// 已中止 — 等待 Reset，支援 Resume
METHOD M_STATE_ABORTED
VAR_INPUT
END_VAR
IF NOT _bRetry THEN
	Busy 	:= FALSE;
	Aborted := TRUE;
	Error 	:= TRUE;
	Status 	:= strStatus;
	_AbortCompleted := FALSE;
	uiAbortingStep  := 0;
END_IF
// 等待上層 FB 設定 Reset
IF reset THEN
	_bRetry := TRUE;
	Busy 	:= FALSE;
	Aborted := FALSE;
	Error 	:= FALSE;
END_IF

IF NOT Execute THEN
	eState := STATE_RESETTING;
END_IF

IF Execute AND _bRetry AND NOT StorageRobot._DI1.Error AND NOT StorageRobot.Halt THEN
	status := '';
	uiExecutingStep := uiResumeStep;
	eState := STATE_EXECUTING;
END_IF
END_METHOD

// 中止 — 停止手臂/馬達/氣缸，保存 Resume 步驟
METHOD M_STATE_ABORTING
VAR_INPUT
END_VAR
CASE uiAbortingStep OF
0:
	// 保存 Resume
	IF uiResumeStep = 0 THEN
		uiResumeStep := uiExecutingStep;
	END_IF
	_Abort	:= FALSE;
	_bRetry := FALSE;

	// 清除 Timer
	TON_TimeOut.IN := FALSE;
	TON_ConveyorTimeOut.IN := FALSE;
	TON_RobotResetTimeOut.IN := FALSE;
	tonDelay_SameSizeGetBox.IN := FALSE;
	tonDelay_SameSizeDelayBox.IN := FALSE;
	uiSameGetBoxStep := 0;

	// 停止手臂 + 倉儲 + NG + PullOut
	//StorageRobot.M_ResetAllCommand();		續做盡量不要清除掉手臂的command 保持原狀，如要清除把Continue 拔掉即可。
	WareHouse.M_ResetFeedInBox();
	NGRegionMove.Execute := FALSE;
	PullOutRegionMove.Execute := FALSE;

	// Phase 2:清 local intent (A00 在 Busy 時 propagate FALSE,本 instance 收手不影響別人)
	bIntent_NeedBackward := FALSE;
	bIntent_HoldStill    := FALSE;

	uiAbortingStep := 100;

100:
	// 機構復位
	uiAbortingStep := 9999;
9999:
	_AbortCompleted := TRUE;
END_CASE

IF NOT Execute THEN
	estate := STATE_RESETTING;
ELSIF _AbortCompleted THEN
	eState := STATE_Aborted;
END_IF
END_METHOD

METHOD M_STATE_DONE
VAR_INPUT
END_VAR
Busy := FALSE;
Done := TRUE;

// 等待上層 FB 取消 Execute
IF NOT Execute THEN
	eState := STATE_RESETTING;
END_IF
END_METHOD

METHOD M_STATE_DORMANT
VAR_INPUT
END_VAR
Busy				:= FALSE;
Done				:= FALSE;
Aborted				:= FALSE;
Error				:= FALSE;
ErrorID				:= 0;
Status				:= '';
_ResetCompleted		:= FALSE;
_Error				:= FALSE;
_Executed			:= FALSE;
_Abort				:= FALSE;
uiExecutingStep		:= 0;
uiResettingStep		:= 0;
uiAbortingStep		:= 0;

_UniqueErrorCode	:= '';
_bRetry				:= FALSE;
uiResumeStep		:= 0;

bBoxA_Done			:= FALSE;
bBoxB_Done			:= FALSE;
bBoxReady			:= FALSE;
bDualGrip			:= FALSE;
bFirstClampIsA		:= TRUE;

TON_TimeOut.IN			:= FALSE;
TON_ConveyorTimeOut.IN	:= FALSE;
TON_RobotResetTimeOut.IN := FALSE;
TON_ArrivedDelay.IN		:= FALSE;
tonDelay_SameSizeGetBox.IN	:= FALSE;
tonDelay_SameSizeDelayBox.IN := FALSE;
uiSameGetBoxStep		:= 0;
tonErrorResetDelay.IN	:= FALSE;
bErrorBlinking			:= FALSE;

PullOutRegionMove.Execute := FALSE;
NGRegionMove.Execute      := FALSE;

// Phase 2:DORMANT 只清 local intent,不動 shared SameSizeCVRequest flag (本 FB 有兩個 instance,idle 不能 stomp 其他 instance 的 request)
bIntent_NeedBackward := FALSE;
bIntent_HoldStill    := FALSE;

_AbortCompleted		:= FALSE;

// 由上層 FB 設定 Execute := TRUE 觸發
IF Execute AND NOT Stop THEN
	// 啟動前檢查
	IF NOT bBoxA_Enable AND NOT bBoxB_Enable THEN
		strStatus := 'No box enabled';
		_UniqueErrorCode := 'E_NO_BOX';
		_Abort := TRUE;
		RETURN;
	END_IF

	// 判斷爪模式
	bDualGrip := bBoxA_Enable AND bBoxB_Enable;
	IF bBoxA_Enable THEN
		bFirstClampIsA := TRUE;
	ELSIF bBoxB_Enable THEN
		bFirstClampIsA := FALSE;
	END_IF

	eState := STATE_EXECUTING;
END_IF
END_METHOD

METHOD M_STATE_ERROR
VAR_INPUT
END_VAR
Busy := FALSE;
Error := TRUE;
Status := strStatus;

// Reset 上升緣 → 1 秒閃爍 (對齊 FB_ShippingRobotTransfer)
trigErrorReset(CLK := Reset);
IF trigErrorReset.Q THEN
	bErrorBlinking := TRUE;
END_IF
tonErrorResetDelay(IN := bErrorBlinking, PT := T#1S);
IF tonErrorResetDelay.Q THEN
	bErrorBlinking := FALSE;
END_IF
IF bErrorBlinking THEN
	Error := FALSE;
END_IF

IF NOT Execute THEN
	Error := FALSE;
	bErrorBlinking := FALSE;
	tonErrorResetDelay.IN := FALSE;
	eState := STATE_RESETTING;
ELSIF trigErrorReset.Q AND Execute AND NOT StorageRobot._DI1.Error THEN
	// Retry 對稱:Reset 上升緣 (edge) 才觸發,從 uiResumeStep 續做
	uiExecutingStep := uiResumeStep;
	Status := '';
	Error := FALSE;
	bErrorBlinking := FALSE;
	tonErrorResetDelay.IN := FALSE;
	eState := STATE_EXECUTING;
END_IF
END_METHOD

// 執行主狀態 — 軌道送盒 + 大手臂取盒 + 入倉/NG
// ═══════════════════════════════════════════════════
// Phase 1 (1000-1500): 第一盒送到 NearStorage
// Phase 2 (2000-2100): 大手臂取第一盒
// Phase 3 (3000-3400): 第二盒送到 NearStorage (雙爪)
// Phase 4 (4000-4100): 大手臂取第二盒
// Phase 5 (5000-5600): 放 ClampA (入倉 or NG)
// Phase 6 (6000-6500): 放 ClampB (入倉 or NG)
// Phase 9 (9000-9100): 復位機構
// ═══════════════════════════════════════════════════
METHOD M_STATE_EXECUTING
VAR_INPUT
END_VAR
Busy := TRUE;

// Stop 時暫停 Timeout
IF Stop THEN
	TON_TimeOut.IN := FALSE;
	TON_ConveyorTimeOut.IN := FALSE;
END_IF

CASE uiExecutingStep OF

0:	// 初始化
	bBoxReady := FALSE;
	bBoxA_Done := FALSE;
	bBoxB_Done := FALSE;
	uiExecutingStep := 1000;

{region '=== Phase 1: 第一盒送到 NearStorage ==='}
// 流程: 馬達 backward + 擋盒 state machine (Press3 後壓 + Press4 擋第二盒) → 送到 NearStorage → motor 停
// 擋盒邏輯 ref FB_RobotRegionMove_AllocatedConveyor uiSameGetBoxStep 0/100/200/300/400 (省略 325/350/375 卡盒重推,Reverse 流程 motor 不能 forward)

1000:	// 請求軌道 backward + 初始化擋盒 state machine
	bIntent_NeedBackward := TRUE;
	bIntent_HoldStill    := FALSE;
	Cylinder.List.fbSameSizeCV_Press3.M_Retract();
	Cylinder.List.fbSameSizeCV_Press4.M_Retract();
	uiSameGetBoxStep := 0;
	TON_ConveyorTimeOut.IN := TRUE;
	uiExecutingStep := 1100;

1100:	// 擋盒 state machine
	CASE uiSameGetBoxStep OF
		0:	// 初始位置:兩支 retract
			Cylinder.List.fbSameSizeCV_Press3.M_Retract();
			Cylinder.List.fbSameSizeCV_Press4.M_Retract();
			uiSameGetBoxStep := 100;

		100:	// 等盒到 Detect6 (50ms debounce) → Press3 extend 後壓
			tonDelay_SameSizeGetBox.IN := Input.bSameSizeCV_BoxDetect6_Sensor;
			IF tonDelay_SameSizeGetBox.Q THEN
				Cylinder.List.fbSameSizeCV_Press3.M_Extend();
				uiSameGetBoxStep := 200;
			END_IF

		200:	// 等 NearStorageSensor 穩定 1.5s 確認盒到位
			tonDelay_SameSizeGetBox.IN := FALSE;
			tonDelay_SameSizeDelayBox.IN := Input.bSameSizeCV_BoxNearStorageSensor;
			IF tonDelay_SameSizeDelayBox.Q THEN
				uiSameGetBoxStep := 300;
			END_IF

		300:	// Press4 extend 擋第二盒避免擠進來
			Cylinder.List.fbSameSizeCV_Press4.M_Extend();
			IF Cylinder.List.fbSameSizeCV_Press4.InFrontPosition THEN
				uiSameGetBoxStep := 400;
			END_IF

		400:	// state machine 完成 → 進 1500 motor 停 + final settle
			tonDelay_SameSizeDelayBox.IN := FALSE;
			uiSameGetBoxStep := 0;
			TON_ConveyorTimeOut.IN := FALSE;
			uiExecutingStep := 1500;
	END_CASE
	// state machine 整段 60s timeout 保護
	IF TON_ConveyorTimeOut.Q THEN
		TON_ConveyorTimeOut.IN := FALSE;
		uiResumeStep := 1000;
		strStatus := 'Phase 1 擋盒 state machine timeout';
		_UniqueErrorCode := 'E_BLOCK_TIMEOUT';
		_Abort := TRUE;
	END_IF

1500:	// 軌道 backward 推到 NearStorage final settle (Press3 後壓中, Press4 擋第二盒中)
	TON_ConveyorTimeOut.IN := TRUE;
	TON_ArrivedDelay.IN := Input.bSameSizeCV_BoxNearStorageSensor;
	IF TON_ArrivedDelay.Q THEN
		TON_ConveyorTimeOut.IN := FALSE;
		bIntent_NeedBackward := FALSE;
		bIntent_HoldStill    := TRUE;	// 大手臂取盒前要靜止
		uiExecutingStep := 1600;
	END_IF
	IF TON_ConveyorTimeOut.Q THEN
		bIntent_NeedBackward := FALSE;
		uiResumeStep := 1000;	// retry 從馬達啟動重來
		strStatus := 'Box cross conveyor timeout';
		_UniqueErrorCode := 'E_BOX_CROSS_TIMEOUT';
		_Abort := TRUE;
	END_IF

1600:	// 等待馬達停止
	 TON_ArrivedDelay.IN := FALSE;
	IF Motor.List.TransmitSameSideCV.InStopped THEN
		//uiExecutingStep := 1650;
		uiExecutingStep := 2000;
	END_IF
1650:	// dead code (1600 直接跳 2000),保留以維持原邏輯 — Destination=WareHouse 視同舊 IsOK=TRUE
	 IF eBoxA_Destination = E_ReverseBoxDestination.WareHouse THEN
	  	uiExecutingStep := 2000;
	 ELSE
		uiExecutingStep := 1700;
  	 END_IF
	 
1700:
	TON_TimeOut.IN := TRUE;
	Cylinder.List.fbSameSizeCV_Press4.M_Extend();
	IF Cylinder.List.fbSameSizeCV_Press4.InFrontPosition THEN
		TON_TimeOut.IN := FALSE;
		uiExecutingStep := 1800;
	END_IF
	IF TON_TimeOut.Q THEN
		uiResumeStep := uiExecutingStep;
		strStatus := 'Press4 Extend timeout';
		_UniqueErrorCode := 'E_CYL_TIMEOUT';
		_Abort := TRUE;
	END_IF
1800:
	Cylinder.List.fbSameSizeCV_Press4.M_Retract();
	IF Cylinder.List.fbSameSizeCV_Press4.InRearPosition THEN				
		uiExecutingStep := 2000;
	END_IF
		 
{endregion}

{region '=== Phase 2: 大手臂取第一盒 ==='}

2000:	// Robot AbsMove 取盒
	TON_TimeOut.IN := TRUE;
	IF NOT StorageRobot._DI1.Done THEN
		StorageRobot.M_StartRobotAbsMove(
			GetBox			:= TRUE,
			UseClampA		:= bFirstClampIsA,
			UseClampB		:= FALSE,
			Area			:= E_RobotArea.TransmitCV,
			ClampA_Address	:= PickupPosition,
			ClampB_Address	:= 99,
			BoxReady_1		:= bFirstClampIsA,
			BoxReady_2		:= FALSE);
	ELSE
		TON_TimeOut.IN := FALSE;
		uiExecutingStep := 2100;
	END_IF
	IF TON_TimeOut.Q OR StorageRobot.Error THEN
		uiResumeStep := uiExecutingStep;
		strStatus := 'Robot pick first box timeout';
		_UniqueErrorCode := 'E_BIGARM_TIMEOUT';
		_Abort := TRUE;
	END_IF

2100:	// Reset Robot
	StorageRobot.M_ResetAllCommand();
	IF NOT StorageRobot._DI1.Done THEN
		IF bDualGrip THEN
			uiExecutingStep := 3000;
		ELSE
			uiExecutingStep := 5000;
		END_IF
	END_IF

{endregion}

{region '=== Phase 3: 第二盒送到 NearStorage (雙爪) ==='}
// 流程同 Phase 1:馬達 backward + 擋盒 state machine → 送到 NearStorage → motor 停

3000:	// 請求軌道 backward + 初始化擋盒 state machine (第二盒)
	bIntent_NeedBackward := TRUE;
	bIntent_HoldStill    := FALSE;
	Cylinder.List.fbSameSizeCV_Press3.M_Retract();
	Cylinder.List.fbSameSizeCV_Press4.M_Retract();
	uiSameGetBoxStep := 0;
	TON_ConveyorTimeOut.IN := TRUE;
	uiExecutingStep := 3100;

3100:	// 擋盒 state machine (第二盒) — ref AllocatedConveyor (與 Phase 1 step 1100 對稱)
	CASE uiSameGetBoxStep OF
		0:
			Cylinder.List.fbSameSizeCV_Press3.M_Retract();
			Cylinder.List.fbSameSizeCV_Press4.M_Retract();
			uiSameGetBoxStep := 100;

		100:	// 等盒到 Detect6 (50ms debounce) → Press3 extend
			tonDelay_SameSizeGetBox.IN := Input.bSameSizeCV_BoxDetect6_Sensor;
			IF tonDelay_SameSizeGetBox.Q THEN
				Cylinder.List.fbSameSizeCV_Press3.M_Extend();
				uiSameGetBoxStep := 200;
			END_IF

		200:	// 等 NearStorageSensor 穩定 1.5s
			tonDelay_SameSizeGetBox.IN := FALSE;
			tonDelay_SameSizeDelayBox.IN := Input.bSameSizeCV_BoxNearStorageSensor;
			IF tonDelay_SameSizeDelayBox.Q THEN
				uiSameGetBoxStep := 300;
			END_IF

		300:	// Press4 extend
			Cylinder.List.fbSameSizeCV_Press4.M_Extend();
			IF Cylinder.List.fbSameSizeCV_Press4.InFrontPosition THEN
				uiSameGetBoxStep := 400;
			END_IF

		400:	// 完成 → 進 3500
			tonDelay_SameSizeDelayBox.IN := FALSE;
			uiSameGetBoxStep := 0;
			TON_ConveyorTimeOut.IN := FALSE;
			uiExecutingStep := 3500;
	END_CASE
	IF TON_ConveyorTimeOut.Q THEN
		TON_ConveyorTimeOut.IN := FALSE;
		uiResumeStep := 3000;
		strStatus := 'Phase 3 擋盒 state machine timeout';
		_UniqueErrorCode := 'E_BLOCK_TIMEOUT';
		_Abort := TRUE;
	END_IF

3500:	// 軌道 backward 推到 NearStorage final settle (第二盒)
	TON_ConveyorTimeOut.IN := TRUE;
	TON_ArrivedDelay.IN := Input.bSameSizeCV_BoxNearStorageSensor;
	IF TON_ArrivedDelay.Q THEN
		TON_ConveyorTimeOut.IN := FALSE;
		bIntent_NeedBackward := FALSE;
		bIntent_HoldStill    := TRUE;	// 大手臂取盒前要靜止
		uiExecutingStep := 3600;
	END_IF
	IF TON_ConveyorTimeOut.Q THEN
		bIntent_NeedBackward := FALSE;
		uiResumeStep := 3000;	// retry 從馬達啟動重來
		strStatus := 'Box 2 cross conveyor timeout';
		_UniqueErrorCode := 'E_BOX_CROSS_TIMEOUT';
		_Abort := TRUE;
	END_IF

3600:	// 等待馬達停止
	 TON_ArrivedDelay.IN := FALSE;
	IF Motor.List.TransmitSameSideCV.InStopped THEN
		//uiExecutingStep := 3650;
		uiExecutingStep := 4000;
	END_IF
3650:	// dead code,保留 — Destination=WareHouse 視同舊 IsOK=TRUE
	 IF eBoxB_Destination = E_ReverseBoxDestination.WareHouse THEN
	  	uiExecutingStep := 4000;
	 ELSE
		uiExecutingStep := 3700;
  	 END_IF
	 
3700:
	TON_TimeOut.IN := TRUE;
	Cylinder.List.fbSameSizeCV_Press4.M_Extend();
	IF Cylinder.List.fbSameSizeCV_Press4.InFrontPosition THEN
		TON_TimeOut.IN := FALSE;
		uiExecutingStep := 3800;
	END_IF
	IF TON_TimeOut.Q THEN
		uiResumeStep := uiExecutingStep;
		strStatus := 'Press4 Extend timeout';
		_UniqueErrorCode := 'E_CYL_TIMEOUT';
		_Abort := TRUE;
	END_IF
3800:
	Cylinder.List.fbSameSizeCV_Press4.M_Retract();
	IF Cylinder.List.fbSameSizeCV_Press4.InRearPosition THEN				
		uiExecutingStep := 4000;
	END_IF

{endregion}

{region '=== Phase 4: 大手臂取第二盒 ==='}

4000:	// Robot AbsMove 第二爪
	TON_TimeOut.IN := TRUE;
	IF NOT StorageRobot._DI1.Done THEN
		StorageRobot.M_StartRobotAbsMove(
			GetBox			:= TRUE,
			UseClampA		:= FALSE,
			UseClampB		:= bFirstClampIsA,
			Area			:= E_RobotArea.TransmitCV,
			ClampA_Address	:= 99,
			ClampB_Address	:= PickupPosition,
			BoxReady_1		:= FALSE,
			BoxReady_2		:= bFirstClampIsA);
	ELSE
		TON_TimeOut.IN := FALSE;
		uiExecutingStep := 4100;
	END_IF
	IF TON_TimeOut.Q OR StorageRobot.Error THEN
		uiResumeStep := uiExecutingStep;
		strStatus := 'Robot pick second box timeout';
		_UniqueErrorCode := 'E_BIGARM_TIMEOUT';
		_Abort := TRUE;
	END_IF

4100:	// Reset Robot
	StorageRobot.M_ResetAllCommand();
	IF NOT StorageRobot._DI1.Done THEN
		uiExecutingStep := 5000;
	END_IF

{endregion}

{region '=== Phase 5: 放 ClampA ==='}

5000:	// 清除 Robot 命令
	TON_RobotResetTimeOut.IN := TRUE;
	StorageRobot.M_ResetAllCommand();
	IF NOT StorageRobot._DI1.Done AND
		NOT (StorageRobot._DI1.AbsMoveA OR StorageRobot._DI1.AbsMoveB OR
			 StorageRobot._DI1.WarehouseA OR StorageRobot._DI1.WarehouseB) THEN
		TON_RobotResetTimeOut.IN := FALSE;
		bBoxReady := FALSE;
		IF bBoxA_Enable THEN
			uiExecutingStep := 5100;
		ELSE
			uiExecutingStep := 6000;
		END_IF
	END_IF
	IF TON_RobotResetTimeOut.Q THEN
		uiResumeStep := 5000;
		strStatus := 'Robot reset timeout (phase 5)';
		_UniqueErrorCode := 'E_BIGARM_TIMEOUT';
		_Abort := TRUE;
	END_IF

5100:	// ClampA Destination 三選一
	CASE eBoxA_Destination OF
		E_ReverseBoxDestination.WareHouse:
			uiExecutingStep := 5200;
		E_ReverseBoxDestination.PullOut:
			uiExecutingStep := 5400;
		E_ReverseBoxDestination.NGConveyor:
			uiExecutingStep := 5300;
	ELSE
		uiResumeStep := 5100;
		strStatus := 'Invalid BoxA destination enum';
		_UniqueErrorCode := 'E_INVALID_DEST';
		_Abort := TRUE;
	END_CASE

5200:	// ClampA OK → 入倉
	TON_TimeOut.IN := TRUE;
	stWareHouseCoord.Layer := iBoxA_Level;
	stWareHouseCoord.Slide := iBoxA_Track;
	IF iBoxA_Warehouse = 1 THEN
		WareHouse.M_StartFeedInBox(WareHouseSelect := E_WareHouse.WareHouseA, WarehouseCoordinates := stWareHouseCoord);
		IF WareHouse.bFeedInBox_Completed THEN
			bBoxReady := TRUE;
		END_IF
		StorageRobot.M_StartWareHousePlaceBox_ClampA(
			WareHouseSelect := E_WareHouse.WareHouseA,
			Info := stWareHouseCoord,
			BoxReady_1st := bBoxReady);
	ELSIF iBoxA_Warehouse = 2 THEN
		WareHouse.M_StartFeedInBox(WareHouseSelect := E_WareHouse.WareHouseB, WarehouseCoordinates := stWareHouseCoord);
		IF WareHouse.bFeedInBox_Completed THEN
			bBoxReady := TRUE;
		END_IF
		StorageRobot.M_StartWareHousePlaceBox_ClampA(
			WareHouseSelect := E_WareHouse.WareHouseB,
			Info := stWareHouseCoord,
			BoxReady_1st := bBoxReady);
	ELSE
		uiResumeStep := 5200;
		strStatus := 'Invalid BoxA warehouse value';
		_UniqueErrorCode := 'E_INVALID_WAREHOUSE';
		_Abort := TRUE;
		RETURN;
	END_IF
	IF StorageRobot._DI1.Done THEN
		TON_TimeOut.IN := FALSE;
		bBoxA_Done := TRUE;
		uiExecutingStep := 5500;
	END_IF
	IF TON_TimeOut.Q OR StorageRobot.Error THEN
		uiResumeStep := 5200;
		strStatus := 'ClampA place to warehouse timeout';
		_UniqueErrorCode := 'E_BIGARM_TIMEOUT';
		_Abort := TRUE;
	END_IF

5300:	// ClampA NG → NG區
	NGRegionMove.Info.Get := FALSE;
	NGRegionMove.Info.UseA := TRUE;
	NGRegionMove.Info.UseB := FALSE;
	NGRegionMove.Info.A_Position := NGAreaPosition;
	NGRegionMove.Info.B_Position := 0;
	NGRegionMove.Execute := TRUE;
	uiExecutingStep := 5310;

5310:	// 等待 NG RegionMove 完成
	IF NGRegionMove.Done THEN
		NGRegionMove.Execute := FALSE;
		bBoxA_Done := TRUE;
		uiExecutingStep := 5320;
	END_IF
	IF NGRegionMove.Error OR NGRegionMove.Aborted THEN
		NGRegionMove.Execute := FALSE;
		uiResumeStep := 5300;
		strStatus := 'ClampA NG region move failed';
		_UniqueErrorCode := 'E_BIGARM_TIMEOUT';
		_Abort := TRUE;
	END_IF

5320:	// 等待 DORMANT
	IF NOT NGRegionMove.Busy AND NOT NGRegionMove.Done THEN
		uiExecutingStep := 5600;
	END_IF

5400:	// ClampA PullOut → PullOutConveyor 區 (Side 1=I3_Slide 左, 2=I4_Slide 右)
	IF iBoxA_PullOutSide < 1 OR iBoxA_PullOutSide > 2 THEN
		uiResumeStep := 5400;
		strStatus := 'Invalid BoxA PullOut side (must be 1 or 2)';
		_UniqueErrorCode := 'E_INVALID_PULLOUT_SIDE';
		_Abort := TRUE;
	ELSE
		PullOutRegionMove.Info.Get := FALSE;
		PullOutRegionMove.Info.UseA := TRUE;
		PullOutRegionMove.Info.UseB := FALSE;
		PullOutRegionMove.Info.A_Position := iBoxA_PullOutSide;
		PullOutRegionMove.Info.B_Position := 0;
		PullOutRegionMove.Execute := TRUE;
		uiExecutingStep := 5410;
	END_IF

5410:	// 等待 PullOut RegionMove 完成
	IF PullOutRegionMove.Done THEN
		PullOutRegionMove.Execute := FALSE;
		bBoxA_Done := TRUE;
		uiExecutingStep := 5420;
	END_IF
	IF PullOutRegionMove.Error OR PullOutRegionMove.Aborted THEN
		PullOutRegionMove.Execute := FALSE;
		uiResumeStep := 5400;
		strStatus := 'ClampA PullOut region move failed';
		_UniqueErrorCode := 'E_BIGARM_TIMEOUT';
		_Abort := TRUE;
	END_IF

5420:	// 等待 DORMANT
	IF NOT PullOutRegionMove.Busy AND NOT PullOutRegionMove.Done THEN
		uiExecutingStep := 5600;
	END_IF

5500:	// ClampA OK 完成 → Reset
	StorageRobot.M_ResetAllCommand();
	WareHouse.M_ResetFeedInBox();
	IF NOT StorageRobot._DI1.Done THEN
		uiExecutingStep := 5600;
	END_IF

5600:	// 繼續 ClampB?
	IF bDualGrip THEN
		bBoxReady := FALSE;
		uiExecutingStep := 6000;
	ELSE
		uiExecutingStep := 9000;
	END_IF

{endregion}

{region '=== Phase 6: 放 ClampB ==='}

6000:	// 準備放 ClampB
	TON_RobotResetTimeOut.IN := TRUE;
	StorageRobot.M_ResetAllCommand();
	IF NOT StorageRobot._DI1.Done AND
		NOT (StorageRobot._DI1.AbsMoveA OR StorageRobot._DI1.AbsMoveB OR
			 StorageRobot._DI1.WarehouseA OR StorageRobot._DI1.WarehouseB) THEN
		TON_RobotResetTimeOut.IN := FALSE;
		uiExecutingStep := 6100;
	END_IF
	IF TON_RobotResetTimeOut.Q THEN
		uiResumeStep := 6000;
		strStatus := 'Robot reset timeout (phase 6)';
		_UniqueErrorCode := 'E_BIGARM_TIMEOUT';
		_Abort := TRUE;
	END_IF

6100:	// ClampB Destination 三選一
	CASE eBoxB_Destination OF
		E_ReverseBoxDestination.WareHouse:
			uiExecutingStep := 6200;
		E_ReverseBoxDestination.PullOut:
			uiExecutingStep := 6400;
		E_ReverseBoxDestination.NGConveyor:
			uiExecutingStep := 6300;
	ELSE
		uiResumeStep := 6100;
		strStatus := 'Invalid BoxB destination enum';
		_UniqueErrorCode := 'E_INVALID_DEST';
		_Abort := TRUE;
	END_CASE

6200:	// ClampB OK → 入倉
	TON_TimeOut.IN := TRUE;
	stWareHouseCoord.Layer := iBoxB_Level;
	stWareHouseCoord.Slide := iBoxB_Track;
	IF iBoxB_Warehouse = 1 THEN
		WareHouse.M_StartFeedInBox(WareHouseSelect := E_WareHouse.WareHouseA, WarehouseCoordinates := stWareHouseCoord);
		IF WareHouse.bFeedInBox_Completed THEN
			bBoxReady := TRUE;
		END_IF
		StorageRobot.M_StartWareHousePlaceBox_ClampB(
			WareHouseSelect := E_WareHouse.WareHouseA,
			Info := stWareHouseCoord,
			BoxReady_2nd := bBoxReady);
	ELSIF iBoxB_Warehouse = 2 THEN
		WareHouse.M_StartFeedInBox(WareHouseSelect := E_WareHouse.WareHouseB, WarehouseCoordinates := stWareHouseCoord);
		IF WareHouse.bFeedInBox_Completed THEN
			bBoxReady := TRUE;
		END_IF
		StorageRobot.M_StartWareHousePlaceBox_ClampB(
			WareHouseSelect := E_WareHouse.WareHouseB,
			Info := stWareHouseCoord,
			BoxReady_2nd := bBoxReady);
	ELSE
		uiResumeStep := 6200;
		strStatus := 'Invalid BoxB warehouse value';
		_UniqueErrorCode := 'E_INVALID_WAREHOUSE';
		_Abort := TRUE;
		RETURN;
	END_IF
	IF StorageRobot._DI1.Done THEN
		TON_TimeOut.IN := FALSE;
		bBoxB_Done := TRUE;
		uiExecutingStep := 6500;
	END_IF
	IF TON_TimeOut.Q OR StorageRobot.Error THEN
		uiResumeStep := 6200;
		strStatus := 'ClampB place to warehouse timeout';
		_UniqueErrorCode := 'E_BIGARM_TIMEOUT';
		_Abort := TRUE;
	END_IF

6300:	// ClampB NG → NG區
	NGRegionMove.Info.Get := FALSE;
	NGRegionMove.Info.UseA := FALSE;
	NGRegionMove.Info.UseB := TRUE;
	NGRegionMove.Info.A_Position := 0;
	NGRegionMove.Info.B_Position := NGAreaPosition;
	NGRegionMove.Execute := TRUE;
	uiExecutingStep := 6310;

6310:	// 等待 NG 完成
	IF NGRegionMove.Done THEN
		NGRegionMove.Execute := FALSE;
		bBoxB_Done := TRUE;
		uiExecutingStep := 6320;
	END_IF
	IF NGRegionMove.Error OR NGRegionMove.Aborted THEN
		NGRegionMove.Execute := FALSE;
		uiResumeStep := 6300;
		strStatus := 'ClampB NG region move failed';
		_UniqueErrorCode := 'E_BIGARM_TIMEOUT';
		_Abort := TRUE;
	END_IF

6320:	// 等待 DORMANT
	IF NOT NGRegionMove.Busy AND NOT NGRegionMove.Done THEN
		uiExecutingStep := 9000;
	END_IF

6400:	// ClampB PullOut → PullOutConveyor 區 (Side 1=I3_Slide 左, 2=I4_Slide 右)
	IF iBoxB_PullOutSide < 1 OR iBoxB_PullOutSide > 2 THEN
		uiResumeStep := 6400;
		strStatus := 'Invalid BoxB PullOut side (must be 1 or 2)';
		_UniqueErrorCode := 'E_INVALID_PULLOUT_SIDE';
		_Abort := TRUE;
	ELSE
		PullOutRegionMove.Info.Get := FALSE;
		PullOutRegionMove.Info.UseA := FALSE;
		PullOutRegionMove.Info.UseB := TRUE;
		PullOutRegionMove.Info.A_Position := 0;
		PullOutRegionMove.Info.B_Position := iBoxB_PullOutSide;
		PullOutRegionMove.Execute := TRUE;
		uiExecutingStep := 6410;
	END_IF

6410:	// 等待 PullOut 完成
	IF PullOutRegionMove.Done THEN
		PullOutRegionMove.Execute := FALSE;
		bBoxB_Done := TRUE;
		uiExecutingStep := 6420;
	END_IF
	IF PullOutRegionMove.Error OR PullOutRegionMove.Aborted THEN
		PullOutRegionMove.Execute := FALSE;
		uiResumeStep := 6400;
		strStatus := 'ClampB PullOut region move failed';
		_UniqueErrorCode := 'E_BIGARM_TIMEOUT';
		_Abort := TRUE;
	END_IF

6420:	// 等待 DORMANT
	IF NOT PullOutRegionMove.Busy AND NOT PullOutRegionMove.Done THEN
		uiExecutingStep := 9000;
	END_IF

6500:	// ClampB OK 完成 → Reset
	StorageRobot.M_ResetAllCommand();
	WareHouse.M_ResetFeedInBox();
	IF NOT StorageRobot._DI1.Done THEN
		uiExecutingStep := 9000;
	END_IF

{endregion}

{region '=== Phase 9: 復位 ==='}

9000:	// 復位機構 (Phase 2:清 local intent,Busy 仍 TRUE 時 A00 會 propagate FALSE)
	bIntent_NeedBackward := FALSE;
	bIntent_HoldStill    := FALSE;
	Cylinder.List.fbSameSizeCV_Press3.M_Retract();
	Cylinder.List.fbSameSizeCV_Press4.M_Retract();
	uiExecutingStep := 9100;

9100:	// 等待復位完成 (Press3 + Press4 縮回 + 馬達停)
	TON_TimeOut.IN := TRUE;
	IF Cylinder.List.fbSameSizeCV_Press3.InRearPosition AND
	   Cylinder.List.fbSameSizeCV_Press4.InRearPosition AND
	   Motor.List.TransmitSameSideCV.InStopped THEN
		TON_TimeOut.IN := FALSE;
		_Executed := TRUE;
	END_IF
	IF TON_TimeOut.Q THEN
		uiResumeStep := uiExecutingStep;
		strStatus := 'Mechanism reset timeout';
		_UniqueErrorCode := 'E_CYL_TIMEOUT';
		_Abort := TRUE;
	END_IF

{endregion}

END_CASE

// 狀態切換
IF _Error THEN
	eState := STATE_ERROR;
ELSIF _Abort THEN
	eState := STATE_ABORTING;
ELSIF _Executed THEN
	eState := STATE_DONE;
ELSIF NOT Execute THEN
	eState := STATE_RESETTING; 
END_IF
END_METHOD

METHOD M_STATE_RESETTING
VAR_INPUT
END_VAR
Busy := TRUE;
Error := FALSE;
Aborted := FALSE;

CASE uiResettingStep OF
0:
	TON_TimeOut.IN := FALSE;
	TON_ConveyorTimeOut.IN := FALSE;
	TON_RobotResetTimeOut.IN := FALSE;
	tonDelay_SameSizeGetBox.IN := FALSE;
	tonDelay_SameSizeDelayBox.IN := FALSE;
	uiSameGetBoxStep := 0;

	StorageRobot.M_ResetAllCommand();
	WareHouse.M_ResetFeedInBox();
	NGRegionMove.Execute := FALSE;
	PullOutRegionMove.Execute := FALSE;
	// Phase 2:清 local intent (Busy=FALSE A00 不會寫,不影響別 instance shared flag)
	bIntent_NeedBackward := FALSE;
	bIntent_HoldStill    := FALSE;

	uiResettingStep := 100;

100:
	Done := FALSE;
	Busy := FALSE;
	_ResetCompleted := TRUE;
END_CASE

IF _ResetCompleted THEN
	eState := STATE_DORMANT;
END_IF
END_METHOD

END_FUNCTION_BLOCK

// ---- Library/20_MachineUnits/22_AllocateArea/Service/FB_PullOutConveyorAction.TcPOU
FUNCTION_BLOCK FB_PullOutConveyorAction EXTENDS FB_ObjectBase_V2 IMPLEMENTS IBasicElement
VAR_INPUT
    FixCylinderA1    : REFERENCE TO FB_Cylinder; // Conveyor A-side 1st cylinder
    FixCylinderA2    : REFERENCE TO FB_Cylinder; // Conveyor A-side 2nd cylinder
    FixCylinderB1    : REFERENCE TO FB_Cylinder; // Conveyor B-side 1st cylinder
    FixCylinderB2    : REFERENCE TO FB_Cylinder; // Conveyor B-side 2nd cylinder
    BarrierCylinderA : REFERENCE TO FB_Cylinder; // Conveyor A-side Barrier cylinder
    BarrierCylinderB : REFERENCE TO FB_Cylinder; // Conveyor B-side Barrier cylinder
    ConveyorMotorA    : REFERENCE TO FB_Motor; // PullOut Conveyor Motor 
	ConveyorMotorB	 : REFERENCE TO FB_Motor; //  Add New Motor Iomapping  edit Min 20250408
	INPUT            : REFERENCE TO ST_InputTable;	
    PullOutInfo      : ST_PullOutConveyorInfo;
END_VAR
VAR_OUTPUT
END_VAR
VAR
	FeedInSensor_A   : BOOL; // PullOut Conveyor A-side FeedIn Sensor
    FeedOutSensor_A  : BOOL; // PullOut Conveyor A-side FeedOut sensor
    DetactSensor_A   : BOOL; // PullOut Conveyor A-side detact sensor
    FeedInSensor_B   : BOOL; // PullOut Conveyor B-side FeedIn Sensor
    FeedOutSensor_B  : BOOL; // PullOut Conveyor B-side FeedOut sensor
    DetactSensor_B   : BOOL; // PullOut Conveyor B-side detact sensor
    TON_MotorRun     : TON; // Pull out conveyor motor running timer.
	TON_MotorReverse : TON; // Pull out conveyor motor reverse timer.
    TON_ForceForward : TON; // When auto process on, the time of force running in command direction.
	TON_MotorStopDelay : TON; // When Conveyor motor stop, the motor will be stopped later, so we need to give a time delay. 
    TON_BoxArrivedDelay: TON; // Check Box arrived(BoxA and BoxB) and delay.
	TON_BarryDelay : TON;
	tonFeedOutTimeOut :TON;
	tonMotorBReverse :TON;
	tonSensorDetectDelay : TON;
	TON_FeedInsensorADelay	:TON;
	TON_betweenboxReverse 	:TON;
	TON_PullOutTimeOut		:TON;
//	_Abort           : BOOL;
	bError			 : BOOL;
	strStatus	     : STRING;
	_UniqueErrorCode : STRING;
	PreviousStrStatus : STRING;
	PreviousErrorCode : STRING;
	
	uiResumeStep	: UINT;
	_bRetry	: BOOL;
END_VAR

A00_BasicUnits();
A10_StateControl();

ACTION A00_BasicUnits:
TON_MotorRun		(PT	:= PullOutInfo.ConveyorRunningTime);
TON_MotorReverse	(PT	:= PullOutInfo.ConveyorReverseTime);
TON_ForceForward	(PT	:= T#0.5S);
TON_MotorStopDelay	(PT := PullOutInfo.ConveyorReverseTime);
TON_BoxArrivedDelay	(PT := T#800MS);
TON_BarryDelay		(PT	:= T#0.1S);
tonFeedOutTimeOut	(PT := PullOutInfo.ConveyorReverseTime*3 );		//notthing use
tonMotorBReverse	(PT := T#1.5S);


tonSensorDetectDelay(PT	:= T#100MS);
TON_FeedInsensorADelay(PT :=T#700MS);
TON_betweenboxReverse(PT :=T#700MS);
TON_PullOutTimeOut (PT :=T#20.0S);



ErrorID := GVL_ErrorCode.GC_SVCID_ALC_PULLOUT_CV;
END_ACTION

ACTION A01_clcExecuting:
FeedInSensor_A  :=INPUT.bPullOutCV_AsideEntry_Sensor;
FeedOutSensor_A  :=INPUT.bPullOutCV_AsideExit_Sensor;
DetactSensor_A   :=input.bPullOutCV_Aside2ndBoxGap_Sensor;
FeedInSensor_B   :=INPUT.bPullOutCV_BsideEntry_Sensor;
FeedOutSensor_B  := INPUT.bPullOutCV_BsideExit_Sensor;
DetactSensor_B   := INPUT.bPullOutCV_Bside2ndBoxGap_Sensor;
END_ACTION

METHOD M_CheckCommand : BOOL
VAR_INPUT
END_VAR
M_CheckCommand := true;
END_METHOD

METHOD M_ResetCylinder : BOOL
VAR_INPUT
END_VAR
END_METHOD

METHOD  M_STATE_ABORTED
VAR_INPUT
END_VAR
IF NOT _bRetry THEN
	Busy 	:= FALSE;
	Aborted := TRUE;
	Error 	:= TRUE;
	Status	:= strStatus;
	uiAbortingStep  := 0;
	_AbortCompleted := FALSE;
	UniqueErrorCode := _UniqueErrorCode;
END_IF
IF reset THEN 
	Aborted := FALSE;
	Error	:= FALSE;
	_bRetry := TRUE;
END_IF


IF NOT Execute THEN
	eState := STATE_RESETTING;
ELSIF Execute AND _bRetry  THEN
	status := '';
	uiExecutingStep := uiResumeStep ;
	eState 			:= STATE_EXECUTING;
END_IF
END_METHOD

METHOD  M_STATE_ABORTING
VAR_INPUT
END_VAR
CASE uiAbortingStep OF
	0:
		_Abort  := FALSE;
		_bRetry := FALSE;
		TON_MotorRun.IN 		:= FALSE;
		tonMotorBReverse.IN 	:= FALSE;
		TON_MotorStopDelay.IN 	:= FALSE;
		
		ConveyorMotorA.M_MotorStop();// .M_StopMotor('Aborting');
		ConveyorMotorB.M_MotorStop();

		uiAbortingStep := 100;
	100:
		IF ConveyorMotorA.InStopped AND ConveyorMotorB.InStopped THEN
			uiAbortingStep := 200;
		END_IF
		
	200:
		uiAbortingStep := 300;
		
	300:
		_AbortCompleted := TRUE;

END_CASE

IF NOT Execute THEN
	eState := STATE_RESETTING;
ELSIF Execute AND _AbortCompleted THEN
	eState := STATE_Aborted;
END_IF
END_METHOD

METHOD  M_STATE_DONE
VAR_INPUT
END_VAR
Busy := FALSE;
Done := TRUE;
//
IF NOT Execute THEN
	eState := STATE_RESETTING;
END_IF
END_METHOD

METHOD  M_STATE_DORMANT
VAR_INPUT
END_VAR
Busy    := FALSE;
Done    := FALSE;
Aborted := FALSE;
Error   := FALSE;
_Error :=FALSE;
ErrorID := 0;
Status  := '';
uiExecutingStep := 0;
uiResettingStep := 0;
uiAbortingStep :=0;
_Abort := FALSE;
_Executed := FALSE;
_ResetCompleted := FALSE;
TON_MotorRun.IN := FALSE;
TON_MotorReverse.IN := FALSE;
TON_ForceForward.IN := FALSE;
TON_MotorStopDelay.IN := FALSE;
TON_BoxArrivedDelay.IN := FALSE;
tonFeedOutTimeOut.IN :=FALSE;
tonMotorBReverse.IN :=FALSE;
tonSensorDetectDelay.IN:=FALSE;

TON_FeedInsensorADelay.IN :=FALSE;
TON_betweenboxReverse.IN :=FALSE;
TON_PullOutTimeOut.IN :=FALSE;
PreviousStrStatus			 :='';
PreviousErrorCode			 :='';
uiResumeStep 	:= 0;
uiAbortingStep  := 0;
_AbortCompleted := FALSE;
_bRetry 		:= false;
//DAS.fbStorageArea.M_InactivePulloutConveyorInternCtrl();
IF Execute THEN
	eState := STATE_EXECUTING;
END_IF
END_METHOD

METHOD  M_STATE_ERROR
VAR_INPUT
END_VAR

Status :=strStatus;
Error:=TRUE;
Busy :=FALSE;
Done :=FALSE;
UniqueErrorCode:=_UniqueErrorCode;
ConveyorMotorA.M_MotorStop();
ConveyorMotorB.M_MotorStop();
IF NOT Execute THEN
	eState :=STATE_RESETTING;
END_IF
END_METHOD

METHOD  M_STATE_EXECUTING
VAR_INPUT
END_VAR
VAR_INST	
END_VAR
Busy := TRUE;
A01_clcExecuting();
CASE uiExecutingStep OF
    0:
        // 非自動模式直接報錯 (避免軸控衝突)
        IF GVL_Machine.PackTags[UnitNo.Allocate].Status.UnitModeCurrent <> E_UnitMode.Auto THEN
            strStatus := 'FB_PullOutConveyorAction Step 0: Not in Auto mode';
            _UniqueErrorCode := 'E_NOT_AUTO_MODE';
            _Error := TRUE;
        ELSE
            IF M_CheckCommand() THEN
                uiExecutingStep := 100;
            ELSE
                Status := 'FB_PullOutConveyorAction Step 0: Wrong command, check the command setting';
                _Error := TRUE;
            END_IF
        END_IF
    100:
        FixCylinderA1.M_Retract();// .M_Retract();//('Clear command');
        FixCylinderA2.M_Retract();//('Clear command');
        FixCylinderB1.M_Retract();//('Clear command');
        FixCylinderB2.M_Retract();//('Clear command');
        BarrierCylinderA.M_Retract();//('Clear command');
        BarrierCylinderB.M_Retract();//('Clear command');

        IF FixCylinderA1.InRearPosition AND
           FixCylinderA2.InRearPosition AND
           FixCylinderB1.InRearPosition AND
           FixCylinderB2.InRearPosition AND
           BarrierCylinderA.InRearPosition AND
           BarrierCylinderB.InRearPosition THEN
            uiExecutingStep := 500;
        END_IF
    500:
        CASE PullOutInfo.CommandType OF
            E_PullOutConveyorCommandType.SideA_FeedIn:
                uiExecutingStep := 1000;
            E_PullOutConveyorCommandType.SideB_FeedIn:
                uiExecutingStep := 2000;
            E_PullOutConveyorCommandType.Both_FeedIn:
                uiExecutingStep := 3000;
            E_PullOutConveyorCommandType.SideA_FeedOut:
                uiExecutingStep := 4000;
            E_PullOutConveyorCommandType.SideB_FeedOut:
                uiExecutingStep := 5000;
            E_PullOutConveyorCommandType.Both_FeedOut:
                uiExecutingStep := 6000;
            E_PullOutConveyorCommandType.MoveForward:
                uiExecutingStep := 7000;
            E_PullOutConveyorCommandType.MoveBackward:
                uiExecutingStep := 8000;
			E_PullOutConveyorCommandType.SlideA_FeedOut_Ext:
				uiExecutingStep := 9000;
			E_PullOutConveyorCommandType.SlideB_FeedOut_Ext:
				uiExecutingStep := 10000;
			E_PullOutConveyorCommandType.SlideA_FeedIn_Ext:
				uiExecutingStep := 11000;
			E_PullOutConveyorCommandType.SlideB_FeedIn_Ext:
				uiExecutingStep := 12000;
        ELSE
            Status := 'FB_PullOutConveyorAction Step 500: Command type out of range.';
            _Error := TRUE;
        END_CASE
		
{region "SideA_FeedIn"}
    1000:
        // Side A feed in box start.
        TON_ForceForward.IN := TRUE;
        ConveyorMotorA.M_MoveForward();// .M_Extend();//;// .M_Extend();//;//('Force forward');

        IF TON_ForceForward.Q THEN
            uiExecutingStep := 1010;
        END_IF
    1010:
        TON_ForceForward.IN := FALSE;
        ConveyorMotorA.M_MotorStop();// .M_MotorStop();//('Force forward stop');
        TON_MotorStopDelay.IN := TRUE;

        IF ConveyorMotorA.InStopped  AND TON_MotorStopDelay.Q THEN
            uiExecutingStep := 1020;
        END_IF
    1020:
        TON_MotorStopDelay.IN := FALSE;
		TON_BoxArrivedDelay.IN := FeedInSensor_A;
        IF TON_BoxArrivedDelay.Q THEN
            uiExecutingStep := 1100;
        ELSE
			TON_BoxArrivedDelay.IN := FALSE;
            uiExecutingStep := 1030;
        END_IF
    1030:
		TON_BoxArrivedDelay.IN := FeedInSensor_A;
        ConveyorMotorA.M_MoveForward();// .M_Extend();//;//('');
        TON_MotorRun.IN := TRUE;

        IF TON_BoxArrivedDelay.Q THEN
            uiExecutingStep := 1100;
        ELSIF TON_MotorRun.Q THEN
            Status := 'FB_PullOutConveyorAction Step 1030: SideA FeedIn no box.';
            _Abort := TRUE;
        END_IF
    1100:
        TON_MotorRun.IN       := FALSE;
        TON_MotorStopDelay.IN := TRUE;
        ConveyorMotorA.M_MotorStop();//('');

        IF ConveyorMotorA.InStopped  AND TON_MotorStopDelay.Q THEN
            uiExecutingStep := 1200;
        END_IF
    1200:
        TON_MotorStopDelay.IN := FALSE;
        FixCylinderA1.M_Extend();// .M_Extend();//('');

        IF FixCylinderA1.InFrontPosition THEN
            uiExecutingStep := 1300;
        END_IF
    1300:
        ConveyorMotorA.M_MoveBackward();// .M_MoveBackward();//('');
        TON_MotorReverse.IN := TRUE;

        IF TON_MotorReverse.Q THEN
            uiExecutingStep := 1400;
        END_IF
    1400:
        ConveyorMotorA.M_MotorStop();//('');
        TON_MotorReverse.IN   := FALSE;
        TON_MotorStopDelay.IN := TRUE;

        IF ConveyorMotorA.InStopped  AND TON_MotorStopDelay.Q THEN
            uiExecutingStep := 1500;
        END_IF
    1500:
        TON_MotorStopDelay.IN := FALSE;
        FixCylinderA1.M_Retract();//('');

        IF FixCylinderA1.InRearPosition THEN
            uiExecutingStep := 99000;
        END_IF

{endregion}

{region "SideB_FeedIn"}
 2000:
        // Side-B feed in start
        TON_ForceForward.IN := TRUE;
        ConveyorMotorB.M_MoveForward(); //('Force forward');

        IF TON_ForceForward.Q THEN
            uiExecutingStep := 2010;
        END_IF
    2010:
        TON_ForceForward.IN   := FALSE;
        TON_MotorStopDelay.IN := TRUE;
        ConveyorMotorB.M_MotorStop();//('Force forward stop');

        IF ConveyorMotorA.InStopped  AND TON_MotorStopDelay.Q THEN
            uiExecutingStep := 2020;
        END_IF
    2020:
        TON_MotorStopDelay.IN := FALSE;
		TON_BoxArrivedDelay.IN := FeedInSensor_B;
        IF TON_BoxArrivedDelay.Q THEN
            uiExecutingStep := 2100;
        ELSE
			TON_BoxArrivedDelay.IN := FALSE;
            uiExecutingStep := 2030;
        END_IF
    2030:
        ConveyorMotorB.M_MoveForward();// 
        TON_MotorRun.IN := TRUE;
		TON_BoxArrivedDelay.IN := FeedInSensor_B;
        IF TON_BoxArrivedDelay.Q THEN
            uiExecutingStep := 2100;
        ELSIF TON_MotorRun.Q THEN
            Status := 'FB_PullOutConveyorAction Step 2030: SideB FeedIn no box.';
            _Abort := TRUE;
        END_IF
    2100:
        TON_MotorRun.IN       := FALSE;
        TON_MotorStopDelay.IN := TRUE;
        ConveyorMotorB.M_MotorStop();//('');

        IF ConveyorMotorB.InStopped  AND TON_MotorStopDelay.Q THEN
            uiExecutingStep := 2200;
        END_IF
    2200:
        TON_MotorStopDelay.IN := FALSE;
        FixCylinderB1.M_Extend();//('');

        IF FixCylinderB1.InFrontPosition THEN
            uiExecutingStep := 2300;
        END_IF
    2300:
        ConveyorMotorB.M_MoveBackward();//('');
        TON_MotorReverse.IN := TRUE;

        IF TON_MotorReverse.Q THEN
            uiExecutingStep := 2400;
        END_IF
    2400:
        ConveyorMotorB.M_MotorStop();//('');
        TON_MotorReverse.IN   := FALSE;
        TON_MotorStopDelay.IN := TRUE;

        IF ConveyorMotorB.InStopped  AND TON_MotorStopDelay.Q THEN
            uiExecutingStep := 2500;
        END_IF
    2500:
        TON_MotorStopDelay.IN := FALSE;
        FixCylinderB1.M_Retract();//('');

        IF FixCylinderB1.InRearPosition THEN
            uiExecutingStep := 99000;
        END_IF
{endregion}

{region "Both_FeedIn"}

    3000:
        // Both side feed in start
        TON_ForceForward.IN := TRUE;
        ConveyorMotorA.M_MoveForward();// ('Force forward');
		ConveyorMotorB.M_MoveForward();// 

        IF TON_ForceForward.Q THEN
            uiExecutingStep := 3010;
        END_IF
    3010:
        TON_ForceForward.IN   := FALSE;
        TON_MotorStopDelay.IN := TRUE;
        ConveyorMotorA.M_MotorStop();//('Force forward stop');
		ConveyorMotorB.M_MotorStop();//('Force forward stop');
		
        IF ConveyorMotorA.InStopped  AND ConveyorMotorB.InStopped  AND TON_MotorStopDelay.Q THEN
            uiExecutingStep := 3020;
        END_IF
    3020:
        TON_MotorStopDelay.IN := FALSE;
		ConveyorMotorA.M_MoveForward();//('Force forward');
		ConveyorMotorB.M_MoveForward();//;//('Force forward');
		
		TON_BoxArrivedDelay.IN := FeedInSensor_A AND FeedInSensor_B;
        IF TON_BoxArrivedDelay.Q THEN
            uiExecutingStep := 3100;
        ELSE
			TON_BoxArrivedDelay.IN := FALSE;
            uiExecutingStep := 3030;
        END_IF
    3030:
        ConveyorMotorA.M_MoveForward();//;//('');
		ConveyorMotorB.M_MoveForward();//;//('');
        TON_MotorRun.IN := TRUE;
		TON_BoxArrivedDelay.IN := FeedInSensor_A AND FeedInSensor_B;
        IF  TON_BoxArrivedDelay.Q THEN
            uiExecutingStep := 3100;
        ELSIF TON_MotorRun.Q THEN
            Status := 'FB_PullOutConveyorAction Step 3030: SideA or SideB FeedIn no box.';
            _Abort := TRUE;
        END_IF
    3100:
        TON_MotorRun.IN       := FALSE;
        TON_MotorStopDelay.IN := TRUE;
        ConveyorMotorA.M_MotorStop();//('');
		ConveyorMotorB.M_MotorStop();//('');
		

        IF ConveyorMotorA.InStopped  AND ConveyorMotorB.InStopped  AND TON_MotorStopDelay.Q THEN
            uiExecutingStep := 3200;
        END_IF
    3200:
        TON_MotorStopDelay.IN := FALSE;
        FixCylinderB1.M_Extend();//('');
        FixCylinderA1.M_Extend();//('');

        IF FixCylinderA1.InFrontPosition AND FixCylinderB1.InFrontPosition THEN
            uiExecutingStep := 3300;
        END_IF
    3300:
        ConveyorMotorA.M_MoveBackward();//('');
		ConveyorMotorB.M_MoveBackward();//('');
        TON_MotorReverse.IN := TRUE;

        IF TON_MotorReverse.Q THEN
            uiExecutingStep := 3400;
        END_IF
    3400:
        ConveyorMotorA.M_MotorStop();//('');
		ConveyorMotorB.M_MotorStop();//('');
        TON_MotorReverse.IN   := FALSE;
        TON_MotorStopDelay.IN := TRUE;

        IF ConveyorMotorA.InStopped  AND ConveyorMotorB.InStopped  AND TON_MotorStopDelay.Q THEN
            uiExecutingStep := 3500;
        END_IF
    3500:
        FixCylinderA1.M_Retract();//('');
        FixCylinderB1.M_Retract();//('');

        IF FixCylinderA1.InRearPosition AND FixCylinderB1.InRearPosition THEN
            uiExecutingStep := 99000;
        END_IF			 
{endregion}

{region "SideA_FeedOut"}
    4000:	//SideA_FeedOut
        ConveyorMotorA.M_MoveBackward();//('');
        TON_MotorReverse.IN := TRUE;

        IF TON_MotorReverse.Q AND NOT FeedInSensor_A THEN
            uiExecutingStep := 4500;
        END_IF
    4500:
        ConveyorMotorA.M_MotorStop();//('');
        TON_MotorReverse.IN   := FALSE;
        TON_MotorStopDelay.IN := TRUE;

        IF ConveyorMotorA.InStopped  AND TON_MotorStopDelay.Q THEN
            uiExecutingStep := 99000;
        END_IF
{endregion}

{region "SideB_FeedOut"}
    5000:	//SideB_FeedOut
        ConveyorMotorB.M_MoveBackward();//('');
        TON_MotorReverse.IN   := TRUE;
        TON_MotorStopDelay.IN := FALSE;

        IF TON_MotorReverse.Q AND NOT FeedInSensor_B THEN
            uiExecutingStep := 5500;
        END_IF
    5500:
        ConveyorMotorB.M_MotorStop();//('');
        TON_MotorReverse.IN   := FALSE;
        TON_MotorStopDelay.IN := TRUE;

        IF ConveyorMotorB.InStopped  AND TON_MotorStopDelay.Q THEN
            uiExecutingStep := 99000;
        END_IF
{endregion}

{region "Both_FeedOut"}
    6000:	//Both_FeedOut
        ConveyorMotorA.M_MoveBackward();//('');
		ConveyorMotorB.M_MoveBackward();//('');
        TON_MotorReverse.IN   := TRUE;
        TON_MotorStopDelay.IN := FALSE;

        IF TON_MotorReverse.Q AND NOT FeedInSensor_A AND NOT FeedInSensor_B THEN
            uiExecutingStep := 6500;
        END_IF
    6500:
        ConveyorMotorA.M_MotorStop();//('');
		ConveyorMotorB.M_MotorStop();//('');
        TON_MotorReverse.IN   := FALSE;
        TON_MotorStopDelay.IN := TRUE;

        IF ConveyorMotorA.InStopped  AND ConveyorMotorB.InStopped  AND TON_MotorStopDelay.Q THEN
            uiExecutingStep := 99000;
        END_IF			 
{endregion}

{region "MoveForward"}
    7000:
        // Move forward start
        ConveyorMotorA.M_MoveForward();//;//('Move forward');
		ConveyorMotorB.M_MoveForward();//;//('Move forward');
        TON_MotorRun.IN := TRUE;
        uiExecutingStep := 7100;
    7100:
        IF TON_MotorRun.Q THEN
            ConveyorMotorA.M_MotorStop();//('Stop');
			ConveyorMotorB.M_MotorStop();//('Stop');
            uiExecutingStep := 7200;
        END_IF
    7200:
        TON_MotorRun.IN       := FALSE;
        TON_MotorStopDelay.IN := TRUE;

        IF ConveyorMotorA.InStopped  AND ConveyorMotorB.InStopped  AND TON_MotorStopDelay.Q THEN
            uiExecutingStep := 99000;
        END_IF
{endregion}

{region "MoveBackward"}
    8000:
        // Move backward start
        ConveyorMotorA.M_MoveBackward();//('Move backward');
		ConveyorMotorB.M_MoveBackward();//('Move backward');
        TON_MotorReverse.IN := TRUE;
        uiExecutingStep := 8100;
    8100:
        IF TON_MotorReverse.Q THEN
            ConveyorMotorA.M_MotorStop();//('Stop');
			ConveyorMotorB.M_MotorStop();//('Stop');
            uiExecutingStep := 8200;
        END_IF
    8200:
        TON_MotorRun.IN       := FALSE;
        TON_MotorStopDelay.IN := TRUE;

        IF ConveyorMotorA.InStopped  AND ConveyorMotorB.InStopped  AND TON_MotorStopDelay.Q THEN
            uiExecutingStep := 99000;
        END_IF 
{endregion}

{region "SlideA_FeedOut_Ext"}
//	9000: // SlideA_FeedOut_Ext

	9000: //SlideA FeedOut_Ext
			ConveyorMotorA.M_MoveBackward();//('');
			tonMotorBReverse.IN :=TRUE;
			IF tonMotorBReverse.Q THEN
				ConveyorMotorA.M_MotorStop();//('');
				uiExecutingStep :=9100;
			END_IF
	9100:	//check sensor make sure full box behide
			IF ConveyorMotorA.InStopped  THEN
				IF (NOT FeedInSensor_A) AND	(NOT DetactSensor_A) THEN
					uiExecutingStep :=99000;
				ELSIF FeedInSensor_A OR	DetactSensor_A THEN
						 uiResumeStep := 9000;
						_Abort :=TRUE;
						strStatus := M_FormatManagedStatus(
							AlarmId := GVL_ErrorCode.GC_ALARM_ALC_PULLOUT_CV,
							InnerMessage := GVL_ErrorCode.GC_MSG_0103);
				END_IF
			END_IF
{endregion}

{region "SlideB_FeedOut_Ext"}
//	10000: // SlideB_FeedOut_Ext


	//======================	SlideB_FeedOut_Ext =====================
	10000: 
			ConveyorMotorB.M_MoveBackward();//('');
			tonMotorBReverse.IN :=TRUE;
			IF tonMotorBReverse.Q THEN
				ConveyorMotorB.M_MotorStop();//('');
				uiExecutingStep :=10100;
			END_IF
	10100:	//check sensor make sure full box behide
			IF ConveyorMotorB.InStopped  THEN
				IF (NOT FeedInSensor_B) AND (NOT DetactSensor_B) THEN
					uiExecutingStep :=99000;
				ELSIF FeedInSensor_B OR	DetactSensor_B THEN
						 uiResumeStep := 10000;
						_Abort 		  := TRUE;
						strStatus := M_FormatManagedStatus(
							AlarmId := GVL_ErrorCode.GC_ALARM_ALC_PULLOUT_CV,
							InnerMessage := GVL_ErrorCode.GC_MSG_0107);
				END_IF
			END_IF
{endregion}

{region "SlideA_FeedIn_Ext"}
	//=======================	SlideA_FeedIn_Ext	near storage side
	11000: 
		IF 	DetactSensor_A AND FeedInSensor_A THEN
			uiExecutingStep := 11100;
		ELSIF NOT DetactSensor_A AND FeedInSensor_A THEN
			uiExecutingStep := 11200;
		ELSIF DetactSensor_A AND NOT FeedInSensor_A THEN
			uiExecutingStep := 11400;
		ELSIF NOT DetactSensor_A AND NOT FeedInSensor_A THEN
			uiExecutingStep := 11400;
		END_IF
	11100: 	// two sensor on
			// Reversemotor unstill two sensor off
		ConveyorMotorA.M_MoveBackward();//('');
		tonMotorBReverse.IN :=TRUE;
		IF tonMotorBReverse.Q THEN
			tonMotorBReverse.IN :=FALSE;
			ConveyorMotorA.M_MotorStop();//('');
			uiExecutingStep :=11110;
		END_IF
		
	11110:	//wait conveyorA stop
		IF ConveyorMotorA.InStopped  THEN
			uiExecutingStep :=11120;
		END_IF
	11120:	//check two sensor
		IF DetactSensor_A OR FeedInSensor_A THEN
			//_Error :=TRUE;
			strStatus := M_FormatManagedStatus(
				AlarmId := GVL_ErrorCode.GC_ALARM_ALC_PULLOUT_CV,
				InnerMessage := GVL_ErrorCode.GC_MSG_0104);
			Status := strStatus;
			Error := TRUE;
			uiExecutingStep :=50000;	//abort step
		ELSE 
			uiExecutingStep :=11800;
		END_IF
		
	11200:	// FeedinSensor on
			//conveyor forward 
			FixCylinderA2.M_Extend();//('');
			IF  FixCylinderA2.InFrontPosition THEN
				ConveyorMotorA.M_MoveForward();// .M_Extend();//;//('');
				uiExecutingStep := 11840;
			END_IF		
	
	11400:	//two sensor off , need make sure no box in two sensor between 
			// Reverse motor to touch detactSensor , make sure no box 
			ConveyorMotorA.M_MoveBackward();//('');
			TON_betweenboxReverse.IN :=TRUE;
			IF TON_betweenboxReverse.Q THEN
				TON_betweenboxReverse.IN :=FALSE;
				ConveyorMotorA.M_MotorStop();//('');
				uiExecutingStep := 11410;
			END_IF
	11410:
			// wait motor stop
			IF ConveyorMotorA.InStopped  THEN
				uiExecutingStep :=11420;
			END_IF
	11420:	//check sensor
			IF DetactSensor_A THEN
				uiExecutingStep :=11430; // todo sth
			ELSIF NOT DetactSensor_A  THEN
				uiExecutingStep :=11800;
			END_IF 
	11430:	//reversemotor unstill sensor off
			ConveyorMotorA.M_MoveBackward();//('');
			TON_betweenboxReverse.IN :=TRUE;	//use to timeout 0.6s
			IF NOT DetactSensor_A THEN
				ConveyorMotorA.M_MotorStop();//('');
				uiExecutingStep :=11440;
			END_IF
			IF TON_betweenboxReverse.Q THEN
				//_Error :=TRUE;
				strStatus := M_FormatManagedStatus(
					AlarmId := GVL_ErrorCode.GC_ALARM_ALC_PULLOUT_CV,
					InnerMessage := GVL_ErrorCode.GC_MSG_0102);
				Status := strStatus;
				Error := TRUE;
				uiExecutingStep :=50000;
			END_IF
	11440:	//wait motor stop
			IF ConveyorMotorA.InStopped  THEN
				uiExecutingStep :=11800;
			END_IF
			
	11800:	//BlockA forward and motorA forward
			BarrierCylinderA.M_Extend();//('');
			IF BarrierCylinderA.InFrontPosition THEN
				ConveyorMotorA.M_MoveForward();//;//('');
				uiExecutingStep :=11810;
			END_IF
	11810:	//wait box move in sensor and pressbox forward
			TON_PullOutTimeOut.IN 	:=TRUE;		//10S
			tonSensorDetectDelay.IN :=DetactSensor_A;		//100MS
			IF tonSensorDetectDelay.Q THEN
				tonSensorDetectDelay.IN :=FALSE;
				TON_PullOutTimeOut.IN 	:=FALSE;
				FixCylinderA2.M_Extend();//('');
				uiExecutingStep :=11820;
			END_IF
			IF TON_PullOutTimeOut.Q THEN
				//_Error :=TRUE;
				strStatus := M_FormatManagedStatus(
					AlarmId := GVL_ErrorCode.GC_ALARM_ALC_PULLOUT_CV,
					InnerMessage := GVL_ErrorCode.GC_MSG_0105);
				Status := strStatus;
				Error := TRUE;
				uiExecutingStep := 50000;
			END_IF
	11820:	//wait PressboxA2 forward and Blockbox backward 
			IF FixCylinderA2.InFrontPosition THEN
				BarrierCylinderA.M_Retract();//('');
				uiExecutingStep :=11830;
			END_IF
	11830:	//wait blockbox backward
			IF BarrierCylinderA.InRearPosition THEN
				uiExecutingStep :=11840;
			END_IF
	11840:	//delay sensor time
			TON_FeedInsensorADelay.IN := FeedInSensor_A ;
			IF TON_FeedInsensorADelay.Q THEN
				TON_FeedInsensorADelay.IN :=FALSE;
				ConveyorMotorA.M_MotorStop();//('');
				uiExecutingStep :=11850;
			END_IF
	11850:	//wait conveyor stop
			IF ConveyorMotorA.InStopped  THEN
				FixCylinderA1.M_Extend();//('');
				uiExecutingStep :=11860;
			END_IF
	11860:	//wait pressbox cylinder move
			IF FixCylinderA1.InFrontPosition THEN
				FixCylinderA1.M_Retract();//('');
				FixCylinderA2.M_Retract();//('');
				uiExecutingStep :=11870;
			END_IF
	11870:	//done
			IF FixCylinderA1.InRearPosition AND FixCylinderA2.InRearPosition THEN
				uiExecutingStep :=99000;
			END_IF
{endregion}

{region "SlideB_FeedIn_Ext"}
	//===========================	SlideB_FeedIn_Ext

	12000: 
		IF 	DetactSensor_B  AND FeedInSensor_B THEN
			uiExecutingStep := 12100;
		ELSIF NOT DetactSensor_B  AND FeedInSensor_B THEN
			uiExecutingStep := 12200;
		ELSIF DetactSensor_B  AND NOT FeedInSensor_B THEN
			uiExecutingStep := 12400;
		ELSIF NOT DetactSensor_B  AND NOT FeedInSensor_B THEN
			uiExecutingStep := 12400;
		END_IF
	12100: 	// two sensor on
			// Reversemotor unstill two sensor off
		ConveyorMotorB.M_MoveBackward();//('');
		tonMotorBReverse.IN :=TRUE;
		IF tonMotorBReverse.Q THEN
			tonMotorBReverse.IN :=FALSE;
			ConveyorMotorB.M_MotorStop();//('');
			uiExecutingStep :=12110;
		END_IF
		
	12110:	//wait conveyorA stop
		IF ConveyorMotorB.InStopped  THEN
			uiExecutingStep :=12120;
		END_IF
	12120:	//check two sensor
		IF DetactSensor_B OR FeedInSensor_B THEN
			_Error :=TRUE;
			strStatus := M_FormatManagedStatus(
				AlarmId := GVL_ErrorCode.GC_ALARM_ALC_PULLOUT_CV,
				InnerMessage := GVL_ErrorCode.GC_MSG_0108);
			Status := strStatus;
			Error := TRUE;
		ELSE 
			uiExecutingStep :=12800;
		END_IF
		
	12200:	// FeedinSensor on
			//conveyor forward 
			FixCylinderB2.M_Extend();//('');
			IF  FixCylinderB2.InFrontPosition THEN
				ConveyorMotorB.M_MoveForward();// .M_Extend();//;//('');
				uiExecutingStep := 12840;
			END_IF		
	
	12400:	//two sensor off , need make sure no box in two sensor between 
			// Reverse motor to touch detactSensor , make sure no box 
			ConveyorMotorB.M_MoveBackward();//('');
			TON_betweenboxReverse.IN :=TRUE;
			IF TON_betweenboxReverse.Q THEN
				TON_betweenboxReverse.IN :=FALSE;
				ConveyorMotorB.M_MotorStop();//('');
				uiExecutingStep := 12410;
			END_IF
	12410:
			// wait motor stop
			IF ConveyorMotorB.InStopped  THEN
				uiExecutingStep :=12420;
			END_IF
	12420:	//check sensor
			IF DetactSensor_B THEN
				uiExecutingStep :=12430; // todo sth
			ELSIF NOT DetactSensor_B  THEN
				uiExecutingStep :=12800;
			END_IF 
	12430:	//reversemotor unstill sensor off
			ConveyorMotorB.M_MoveBackward();//('');
			TON_betweenboxReverse.IN :=TRUE;	//use to timeout 0.6s
			IF NOT DetactSensor_B THEN
				ConveyorMotorB.M_MotorStop();//('');
				uiExecutingStep :=12440;
			END_IF
			IF TON_betweenboxReverse.Q THEN
				_Error :=TRUE;
				strStatus := M_FormatManagedStatus(
					AlarmId := GVL_ErrorCode.GC_ALARM_ALC_PULLOUT_CV,
					InnerMessage := GVL_ErrorCode.GC_MSG_0106);
				Status := strStatus;
				Error := TRUE;
			END_IF
	12440:	//wait motor stop
			IF ConveyorMotorB.InStopped  THEN
				uiExecutingStep :=12800;
			END_IF
			
	12800:	//BlockA forward and motorA forward
			BarrierCylinderB.M_Extend();//('');
			IF BarrierCylinderB.InFrontPosition THEN
				ConveyorMotorB.M_MoveForward();//;//('');
				uiExecutingStep :=12810;
			END_IF
	12810:	//wait box move in sensor and pressbox forward
			TON_PullOutTimeOut.IN 	:=TRUE;		//10S
			tonSensorDetectDelay.IN :=DetactSensor_B;		//100MS
			IF tonSensorDetectDelay.Q THEN
				tonSensorDetectDelay.IN :=FALSE;
				TON_PullOutTimeOut.IN 	:=FALSE;
				FixCylinderB2.M_Extend();//('');
				uiExecutingStep :=12820;
			END_IF
			IF TON_PullOutTimeOut.Q THEN
				_Error :=TRUE;
				strStatus := M_FormatManagedStatus(
					AlarmId := GVL_ErrorCode.GC_ALARM_ALC_PULLOUT_CV,
					InnerMessage := GVL_ErrorCode.GC_MSG_0105);
				Status := strStatus;
				Error := TRUE;
			END_IF
	12820:	//wait PressboxB2 forward & Blockbox backward 
			IF FixCylinderB2.InFrontPosition THEN
				BarrierCylinderB.M_Retract();//('');
				uiExecutingStep :=12830;
			END_IF
	12830:	//wait blockbox backward
			IF BarrierCylinderB.InRearPosition THEN
				uiExecutingStep :=12840;
			END_IF
	12840:	//delay sensor time
			TON_FeedInsensorADelay.IN := FeedInSensor_B ;
			IF TON_FeedInsensorADelay.Q THEN
				TON_FeedInsensorADelay.IN :=FALSE;
				ConveyorMotorB.M_MotorStop();//('');
				uiExecutingStep :=12850;
			END_IF
	12850:	//wait conveyor stop
			IF ConveyorMotorB.InStopped  THEN
				FixCylinderB1.M_Extend();//('');
				uiExecutingStep :=12860;
			END_IF
	12860:	//wait pressbox cylinder move
			IF FixCylinderB1.InFrontPosition THEN
				FixCylinderB1.M_Retract();//('');
				FixCylinderB2.M_Retract();//('');
				uiExecutingStep :=12870;
			END_IF
	12870:	//done
			IF FixCylinderB1.InRearPosition AND FixCylinderB2.InRearPosition THEN
				uiExecutingStep :=99000;
			END_IF
{endregion}

	50000:	//SlideA FeedIn Ext Resume step
			FixCylinderA1.M_Retract();
			FixCylinderA2.M_Retract();
			BarrierCylinderA.M_Retract();
			ConveyorMotorA.M_MotorStop();
			TON_PullOutTimeOut.IN :=FALSE;
			TON_betweenboxReverse.IN :=FALSE;
			IF FixCylinderA1.InRearPosition AND 
				FixCylinderA2.InRearPosition AND 
				BarrierCylinderA.InRearPosition AND 
				ConveyorMotorA.InStopped THEN
				uiResumeStep := 11000;
				_Abort :=TRUE;
			END_IF
			
    99000:
        TON_MotorStopDelay.IN := FALSE;
        _Executed             := TRUE;

END_CASE

IF _Executed THEN
    eState := STATE_DONE;
ELSIF NOT Execute THEN
    eState := STATE_RESETTING;
ELSIF _Abort OR Abort THEN
    eState := STATE_ABORTING;
ELSIF _Error THEN
	eState:=STATE_ERROR;	
END_IF
END_METHOD

METHOD  M_STATE_RESETTING
VAR_INPUT
END_VAR
CASE uiResettingStep OF
	0:
		FixCylinderA1.M_Retract();// .M_Retract();//('Resetting');
		FixCylinderA2.M_Retract();//('Resetting');
		FixCylinderB1.M_Retract();//('Resetting');
		FixCylinderB2.M_Retract();//('Resetting');
		BarrierCylinderA.M_Retract();//('Resetting');
		BarrierCylinderB.M_Retract();//('Resetting');
		uiResettingStep := 100;
	100:
		IF FixCylinderA1.InRearPosition AND
			FixCylinderA2.InRearPosition AND
			FixCylinderB1.InRearPosition AND
			FixCylinderB2.InRearPosition AND
			BarrierCylinderA.InRearPosition AND 
			BarrierCylinderB.InRearPosition THEN
			uiResettingStep := 200;
		END_IF
	200:
		ConveyorMotorA.M_MotorStop();// .M_StopMotor('Resetting');
		ConveyorMotorB.M_MotorStop();
		uiResettingStep := 300;
	300:
		IF ConveyorMotorA.InStopped AND 
			ConveyorMotorB.InStopped THEN
		//	DAS.fbStorageArea.M_InactivePulloutConveyorInternCtrl();
			uiResettingStep := 9000;
		END_IF
	9000:
		_Error :=false;
		 Error :=false;
		_ResetCompleted := TRUE;
END_CASE
IF _ResetCompleted THEN
	eState := STATE_DORMANT;
END_IF
END_METHOD

END_FUNCTION_BLOCK

// ---- Library/20_MachineUnits/21_StorageArea/Service_Robot/FB_RobotRegionMove_FeedInConveyor_V2.TcPOU
FUNCTION_BLOCK FB_RobotRegionMove_FeedInConveyor_V2 EXTENDS FB_ObjectBase_V2 IMPLEMENTS IBasicElement
VAR_INPUT
    Robot     					: REFERENCE TO FB_FanucRobot_Basic_V2;
	LowerConveyor				: REFERENCE TO FB_Motor;
	Input 						: REFERENCE TO ST_InputTable;

   // Command   : ST_WareHouseWithRobotMove_Command;
    Info	  					: ST_RobotRegionMove_Info;
	Stop	  					: BOOL;
	bCheckUpperCV_ServiceDone	: BOOL;
END_VAR
VAR_OUTPUT
  // Status : ST_WareHouseWithRobotMove_Status;
  
END_VAR
VAR
	//_Abort		: BOOL;
	strStatus	: STRING;
	uiResumeStep : UDINT;
	
	Area	: E_RobotArea := E_RobotArea.InOutConveyor;
	UseA 	: BOOL;
	UseB	: BOOL;
	
	Get 	:BOOL;
	tonTimeOut	:TON;
	bTimeOutIN			   : BOOL;
	tonDelay	 : TON;
	_UniqueErrorCode :STRING;
	PreviousStrStatus : STRING;
	PreviousErrorCode : STRING;
	//Added by Jidien Kachu in 2025/10/09
	uiLastBothStep	: UINT;
	uiLastSingleClampStep	: UINT;
	bRobotTimeOutIN	: BOOL;
	tonRobotTimeOut	: TON;
	uiBothStep	: UINT;
	uiSingleClampStep	: UINT;	
	
	_bRetry	: BOOL;
END_VAR

SUPER^.A10_StateControl();
A00_BasicUnits();

(*============================================================
Create Date : 2025/11/24
Last Update	: 2026/04/01
Change Log  : 2025/11/24，Fix StateControl Switch , the version extend Kachue verion from TH_Mirror DAS // Edited : Gamin
			  2026/04/01，移植泰興鏡射機版本。
============================================================*)

ACTION A00_BasicUnits:
tonTimeOut(IN:= bTimeOutIN AND NOT THIS^.Stop, PT:=T#60S);
tonDelay(PT:=T#1S);
tonRobotTimeOut(IN:= bRobotTimeOutIN AND NOT THIS^.Stop, PT:=T#60S);
ErrorID:=2240;
END_ACTION

METHOD M_CheckCommand : BOOL // True : Command is useful
VAR_INPUT
END_VAR
VAR
	
END_VAR
// Check command paremeter is correct
	
	THIS^.Get :=Info.Get;
	UseA := Info.UseA;
	UseB := Info.UseB;

	 //FeedIn/Out conveyor
	 	IF UseA THEN	 
			IF  (Info.A_Position<1 OR  Info.A_Position>3 )THEN
				strStatus:='FB_RobotRegionMove_FeedInConveyor_V2: Wrong command ,Position A Not allow';
				M_CheckCommand:=FALSE;
				RETURN;	
			ELSIF  Info.A_Position=3 AND Get THEN
				strStatus:='FB_RobotRegionMove_FeedInConveyor_V2: Wrong command ,Can Not Get box from FeedOut conveyor ';
				M_CheckCommand:=FALSE;
				RETURN;
			ELSIF 	Info.A_Position <>3 AND NOT Get THEN
				strStatus:='FB_RobotRegionMove_FeedInConveyor_V2: Wrong command ,Can Not Put box to FeedIn conveyor ';
				M_CheckCommand:=FALSE;
				RETURN;				
			END_IF
		END_IF
		
		IF UseB AND ( Info.B_Position<1 OR  Info.B_Position>3 )THEN
			strStatus:='FB_RobotRegionMove_FeedInConveyor_V2: Wrong command ,Position B Not allow';
			M_CheckCommand:=FALSE;
			RETURN;	
		ELSIF UseB AND Info.B_Position=3 AND Get THEN
			strStatus:='FB_RobotRegionMove_FeedInConveyor_V2: Wrong command ,Can Not Get box from FeedOut conveyor ';
			M_CheckCommand:=FALSE;
			RETURN;		
		ELSIF UseB AND Info.B_Position <>3 AND NOT Get THEN
			strStatus:='FB_RobotRegionMove_FeedInConveyor_V2: Wrong command ,Can Not Put box to FeedIn conveyor ';
			M_CheckCommand:=FALSE;
			RETURN;		
		END_IF
		
M_CheckCommand:=TRUE;
END_METHOD

METHOD M_CheckUnitsNotBusy : BOOL
VAR_INPUT
END_VAR
M_CheckUnitsNotBusy := true;
END_METHOD

METHOD M_CheckUnitsReady : BOOL
VAR_INPUT
END_VAR
M_CheckUnitsReady := true;
END_METHOD

METHOD M_ResetHomingFeedOut : BOOL
VAR_INPUT
END_VAR
Execute := FALSE;
info.UseA := FALSE;
info.UseB := FALSE;

M_ResetHomingFeedOut := TRUE;
END_METHOD

METHOD M_StartHomingFeedOut : BOOL
VAR_INPUT
	UseA	: BOOL;
	UseB	: BOOL;
END_VAR
// NG conveyor homing only place
Info.Get := FALSE;

Info.UseA := UseA;
info.UseB := UseB;

IF UseA AND UseB THEN
	Info.A_Position := 3;
	Info.B_Position := 3;
ELSIF UseA THEN
	Info.A_Position := 3;
	info.B_Position := 99;
ELSIF UseB THEN
	info.A_Position	:= 99;
	Info.B_Position := 3;
END_IF

Execute := TRUE;

M_StartHomingFeedOut := TRUE;
END_METHOD

METHOD  M_STATE_ABORTED
VAR_INPUT
END_VAR
IF NOT _bRetry THEN
	Busy	:= FALSE;
	Error 	:= TRUE;
	Aborted := TRUE;
	Status 	:= strStatus;
	UniqueErrorCode:=_UniqueErrorCode;
	uiAbortingStep := 0;
	_AbortCompleted:=FALSE;//Edited by Jidien Kachu in 2025/10/14
END_IF

IF reset THEN
	_bRetry := TRUE;
	Error 	:= FALSE;
	Aborted := FALSE;
END_IF

IF NOT Execute THEN
	eSTATE:=STATE_RESETTING;
END_IF
IF Execute AND _bRetry AND NOT Robot._DI1.Error AND NOT Robot.Halt THEN
	PreviousStrStatus := strStatus;
	PreviousErrorCode := _UniqueErrorCode;
	uiExecutingStep   := uiResumeStep;
	(* Edited by Jidien Kachu in 2025/10/09 *)
	uiBothStep 		  := uiLastBothStep;
	uiSingleClampStep := uiLastSingleClampStep;

	Status := '';

	(*====================================*)
	IF GVL_ADS.MachineState <>E_MachineState.Error THEN
		eSTATE:=STATE_EXECUTING;
	END_IF
END_IF
END_METHOD

METHOD  M_STATE_ABORTING
VAR_INPUT
END_VAR
CASE uiAbortingStep OF
	0 :
			bTimeOutIN		:= FALSE;
			bRobotTimeOutIN := FALSE;
			tonDelay.IN 	:= FALSE;
			_bRetry:= FALSE;
			_Abort := FALSE;
			
			LowerConveyor.M_MotorStop();
			IF strStatus = PreviousStrStatus THEN
				_UniqueErrorCode :=PreviousErrorCode;
			END_IF
			uiAbortingStep:=100;
	100:		
			 IF DAS_CoreSys.MachineControl.M_RobotResetCmd() THEN
				 uiAbortingStep := 200;
			 END_IF
	200:
			IF DAS_CoreSys.MachineControl.M_RobotStartCmd() THEN
				 uiAbortingStep := 300;
			 END_IF 
	300:
			IF Robot._DI1.Error THEN
		 		uiAbortingStep := 100;
			ELSE
				uiAbortingStep := 9999;
			END_IF
	
	9999:	
			_AbortCompleted:=TRUE;
END_CASE

IF _AbortCompleted THEN	
	eSTATE :=STATE_ABORTED;
END_IF
END_METHOD

METHOD  M_STATE_DONE
VAR_INPUT
END_VAR
Busy   := FALSE;
_Error := Error := FALSE;
_Abort := Abort := FALSE;
Done   := TRUE;

IF NOT Execute THEN
    eState := STATE_RESETTING;
END_IF
END_METHOD

METHOD  M_STATE_DORMANT
VAR_INPUT
END_VAR
// Clear FB output
Busy            := FALSE;
Done            := FALSE;
_Abort			:= FALSE;
Aborted         := FALSE;
Error           := FALSE;
ErrorID         := 0;
Status          := '';
_ResetCompleted := FALSE;
_Error          := FALSE;
_Executed       := FALSE;
tonDelay.IN := FALSE;
bTimeOutIN:=FALSE;
bRobotTimeOutIN := FALSE;
strStatus :='FB_RobotRegionMove_FeedInConveyor_V2: No Error';
uiExecutingStep :=uiResettingStep :=uiResumeStep :=0;
uiBothStep			:= 0; 
uiSingleClampStep 	:= 0;
uiLastBothStep		:= 0; 
uiLastSingleClampStep := 0; 
_UniqueErrorCode :='0';
tonRobotTimeOut.IN := FALSE;
PreviousStrStatus			 :='';
PreviousErrorCode			 :='';
_bRetry				:= FALSE;

// Wait Execute command
IF Execute AND NOT stop THEN
    eState := STATE_EXECUTING;
END_IF
END_METHOD

METHOD  M_STATE_ERROR
VAR_INPUT
END_VAR
ERROR   :=TRUE;
Busy	:=FALSE;
Status := strStatus;
UniqueErrorCode:=_UniqueErrorCode;
IF NOT Execute THEN	
eSTATE:=STATE_RESETTING;
END_IF
END_METHOD

METHOD  M_STATE_EXECUTING
VAR_INPUT
END_VAR
VAR_INST
	BoxReady_1st : BOOL;
	BoxReady_2nd : BOOL;
//    uiBothStep : UINT;
//    uiSingleClampStep : UINT;	
	Address_A : INT;
	Address_B : INT;
END_VAR
VAR
	WareHouse: INT;
END_VAR
// Set Busy active edit by johnson
Busy := TRUE;
(*IF THIS^.Stop THEN // Pending the timeout when Stop signal occur
	bTimeoutIN:=FALSE;
END_IF*)
// Service Process
CASE uiExecutingStep OF
	0:
        // Clear variable
//        uiBothStep := 0;
		uiLastBothStep := 0; //Edited by Jidien Kachu in 2025/10/09
//		uiSingleClampStep :=0;
		uiLastSingleClampStep := 0; //Edited by Jidien Kachu in 2025/10/09
		BoxReady_1st := 0;
		BoxReady_2nd := 0;
		bTimeOutIN:=FALSE;
        // Check command
        IF M_CheckCommand() THEN
            uiExecutingStep := 10;
		ELSE
			_Error:=TRUE;
        END_IF
    10:
        // Start process, check units first
        IF M_CheckUnitsReady() THEN
            uiExecutingStep := 20;
        END_IF
    20:
        // CHeck units not busy state
        IF M_CheckUnitsNotBusy() THEN
            uiExecutingStep := 1000;
        END_IF
   
	1000:   
			// Read   coordinate
			 Area := THIS^.Area;
 			 Address_A := LREAL_TO_INT(Info.A_Position);
			 Address_B := LREAL_TO_INT(Info.B_Position);
			 
			IF UseA AND NOT UseB THEN
				//Only clampA
				uiExecutingStep := 10000;
			ELSIF NOT UseA AND UseB THEN
				//Only ClampB 
				uiExecutingStep := 20000;
			ELSIF UseA AND UseB THEN
				//Both Clamps
				uiExecutingStep := 30000;		
			ELSE
				strStatus := 'FB_RobotRegionMove_FeedInConveyor_V2 Step 1000: No clamp selected';
				_Error 	  := TRUE;
			END_IF

	10000:	// 檢查 A爪 Sensor判斷是否可以安全做動
			IF Get THEN
				IF  Robot._DI1.ClampA_Open THEN		// AClamp has box
					uiExecutingStep := 11000;
				ELSE
					_Error 	  := TRUE;
					strStatus := 'FB_RobotRegionMove_FeedInConveyor_V2 Step 10000: AClamp not open';
				END_IF
			ELSE
				IF NOT Robot._DI1.ClampA_Open THEN	// AClamp has box
					uiExecutingStep := 11000;
				ELSE	
					_Error 	  := TRUE;
					strStatus := 'FB_RobotRegionMove_FeedInConveyor_V2 Step 10000: AClamp is open';
				END_IF
			END_IF
       
    11000: // Only ClampA 
        IF NOT Robot._DI1.Done THEN
            
            
			CASE uiSingleClampStep OF
				
				0://
				
					CASE Address_A OF
						1,2:
							uiSingleClampStep:=1000;
						
						3: 
							uiSingleClampStep:=100;
					END_CASE
				
				100:	
					LowerConveyor.M_MoveBackward();
					tonDelay.IN := FALSE;
					IF ( NOT Input.bLowCV_BoxArrived_Sensor) AND ( Input.bLowCV_2ndBoxGap_Sensor) THEN
						bTimeOutIN:=FALSE;
						uiSingleClampStep:=150;
					END_IF
					bTimeOutIN:=TRUE;
					IF tonTimeOut.Q=TRUE OR Robot._DI1.Error THEN
						strStatus := 'FB_RobotRegionMove_FeedInConveyor_V2 Step 11000: Empty conveyor timeout';
						uiResumeStep:=11000;
						uiLastSingleClampStep := 0; //Edited by Jidien Kachu in 2025/10/09
						uiAbortingStep := 0;//Edited by Jidien Kachu in 2025/10/14
						_Abort:=TRUE;
					END_IF
				150:
					tonDelay.IN := TRUE;
					IF tonDelay.Q THEN
						uiSingleClampStep:=200;
					END_IF	
				200:
					tonDelay.IN := FALSE;
					LowerConveyor.M_MotorStop();
					uiSingleClampStep:=300;
				
				300:
					IF 	LowerConveyor.InStopped THEN
						bTimeOutIN:=FALSE;
						BoxReady_1st:=TRUE;
						uiSingleClampStep:=9999;
					END_IF
					bTimeOutIN:=TRUE;
					IF tonTimeOut.Q=TRUE OR Robot._DI1.Error THEN
						strStatus :='FB_RobotRegionMove_FeedInConveyor_V2 Step 11000: Stop Conveyor timeout';


						(* Edited by Jidien Kachu in 2025/10/09*)
//						_Error:=TRUE;
						uiResumeStep:=11000;
						uiLastSingleClampStep := 200;
						uiAbortingStep := 0;//Edited by Jidien Kachu in 2025/10/14
						_Abort:=TRUE;
						(*===================================*)
					END_IF	
				
				1000:
						CASE Address_A OF
						1:
								IF 	bCheckUpperCV_ServiceDone AND Input.bUpCV_Block1Detect_Sensor THEN
										BoxReady_1st := TRUE;
								END_IF
						2:
								IF 	bCheckUpperCV_ServiceDone AND Input.bUpCV_BoxArrived_Sensor THEN
										BoxReady_1st := TRUE;
								END_IF
						END_CASE						
						
				9999: //
						;
			END_CASE
			          		 
				  // Robot Abs move
           		 Robot.M_StartRobotAbsMove(GetBox:=Get,
											UseClampA:=UseA,
											UseClampB:=UseB,
											Area:=Area,
											ClampA_Address:=Address_A,
											ClampB_Address:=Address_B,
											BoxReady_1:=BoxReady_1st,
											BoxReady_2:=BoxReady_2nd);				  
		
        ELSE
//			bTimeOutIN:=FALSE;
			bRobotTimeOutIN := FALSE; //edited by Jidien Kachu in 2025/10/09
            uiExecutingStep := 10080;
        END_IF
		(* Edited by Jidien Kachu in 2025/10/09*)

		bRobotTimeOutIN := TRUE;

		IF tonRobotTimeOut.Q THEN

			bRobotTimeOutIN := FALSE;
			uiResumeStep 	:= 11000;
			strStatus 		:= 'FB_RobotRegionMove_FeedInConveyor_V2 Step 11000: Robot Abs move timeout';
			_Abort			:= TRUE;
		END_IF	
		IF Robot.Error THEN
			bRobotTimeOutIN := FALSE;
			uiResumeStep 	:= 11000;
			strStatus 		:= CONCAT('FB_RobotRegionMove_FeedInConveyor_V2',robot.ErrMsg);
			_Abort			:= TRUE;
		END_IF
		(*===================================*)
    10080:
        Robot.M_ResetRobotAbsMove(UseA,UseB); // Clear command and go to place box

		bRobotTimeOutIN := TRUE; //Edited by Jidien Kachu in 2025/10/09
        IF NOT Robot._DI1.Done THEN

			bRobotTimeOutIN := FALSE; //Edited by Jidien Kachu in 2025/10/09
            uiExecutingStep := 80000; 
        END_IF
		(* Edited by Jidien Kachu in 2025/10/09 *)

		IF tonRobotTimeOut.Q THEN
			bRobotTimeOutIN := FALSE;
			strStatus 		:= 'FB_RobotRegionMove_FeedInConveyor_V2 Step 10080: Reset Robot timeout';
			_Error:=TRUE;
		END_IF	
		(*=====================================*)
    
	10090: // Check box 

	20000:	// 檢查 B爪 Sensor判斷，是否可以安全做動。
			IF Get THEN
				IF  Robot._DI1.ClampB_Open THEN	// BClamp has box
					uiExecutingStep := 21000;
				ELSE
					_Error	  := TRUE;
					strStatus := 'FB_RobotRegionMove_FeedInConveyor_V2 Step 20000: BClamp not open';
				END_IF
			ELSE
				IF NOT Robot._DI1.ClampB_Open THEN	// BClamp has box
					uiExecutingStep := 21000;
				ELSE
					_Error	  := TRUE;
					strStatus := 'FB_RobotRegionMove_FeedInConveyor_V2 Step 20000: BClamp is open';
				END_IF
			END_IF
		
			
    21000: // Only ClampB
        IF NOT Robot._DI1.Done THEN
			
            	CASE uiSingleClampStep OF
				
				0://
				
					CASE Address_B OF
						1,2:
							uiSingleClampStep:=1000;
						
						3: 
							uiSingleClampStep:=100;
					END_CASE
			
				100:	
					LowerConveyor.M_MoveBackward();
					IF (NOT Input.bLowCV_BoxArrived_Sensor) AND  Input.bLowCV_2ndBoxGap_Sensor THEN
						bTimeOutIN:=FALSE;
						tonDelay.IN := FALSE;
						uiSingleClampStep:=150;
					END_IF
					bTimeOutIN:=TRUE;
					IF tonTimeOut.Q=TRUE OR Robot._DI1.Error THEN
						strStatus 				:= 'FB_RobotRegionMove_FeedInConveyor_V2 Step 21000: Empty conveyor timeout';
						uiResumeStep			:= 21000;
						uiLastSingleClampStep 	:= 0; //Edited by Jidien Kachu in 2025/10/09
						uiAbortingStep 			:= 0;//Edited by Jidien Kachu in 2025/10/14
						_Abort					:= TRUE;
					END_IF
					
				150:
					tonDelay.IN := TRUE;
					IF tonDelay.Q THEN
						uiSingleClampStep:=200;
					END_IF		
				200:
					tonDelay.IN := FALSE;
					LowerConveyor.M_MotorStop();
					uiSingleClampStep:=300;
				
				300:
					IF 	LowerConveyor.InStopped THEN
						bTimeOutIN:=FALSE;
						BoxReady_2nd:=TRUE;
						uiSingleClampStep:=9999;
					END_IF
					bTimeOutIN:=TRUE;
					IF tonTimeOut.Q=TRUE OR Robot._DI1.Error THEN
						strStatus :='FB_RobotRegionMove_FeedInConveyor_V2 Step 21000: Stop Conveyor timeout';




//						_Error:=TRUE;
						(* Edited by Jidien Kachu in 2025/10/09 *)
						uiResumeStep := 21000;
						uiLastSingleClampStep := 200;
						uiAbortingStep := 0;//Edited by Jidien Kachu in 2025/10/14
						_Abort := TRUE;
						(*====================================*)
					END_IF	
				
				1000:

						CASE Address_B OF
						1:
							IF 	bCheckUpperCV_ServiceDone AND Input.bUpCV_Block1Detect_Sensor THEN
								BoxReady_2nd := TRUE;
							END_IF
													
						2:
							IF 	bCheckUpperCV_ServiceDone AND Input.bUpCV_BoxArrived_Sensor THEN
								BoxReady_2nd := TRUE;
							END_IF

						END_CASE						
						
				9999 ://
			END_CASE	
		
			
			          		 
				  // Robot Abs move
           		 Robot.M_StartRobotAbsMove( GetBox:=Get,
											UseClampA:=UseA,
											UseClampB:=UseB,
											Area:=Area,
											ClampA_Address:=Address_A,
											ClampB_Address:=Address_B,
											BoxReady_1:=BoxReady_1st,
											BoxReady_2:=BoxReady_2nd);	
        ELSE
//			bTimeOutIN:=FALSE;
			bRobotTimeOutIN := FALSE; //Edited by Jidien Kachu in 2025/10/09
            uiExecutingStep := 20080;
        END_IF
		(* Edited by Jidien Kachu in 2025/10/09 *)

		bRobotTimeOutIN := TRUE;

		IF tonRobotTimeOut.Q THEN

			bRobotTimeOutIN := FALSE;
			uiResumeStep 	:= 21000;
			strStatus 		:= 'FB_RobotRegionMove_FeedInConveyor_V2 Step 21000: Robot Abs move timeout';
			_Abort			:= TRUE;
		END_IF	
		IF Robot.Error THEN
			bRobotTimeOutIN := FALSE;
			uiResumeStep 	:= 21000;
			strStatus 		:= CONCAT('FB_RobotRegionMove_FeedInConveyor_V2',robot.ErrMsg);
			_Abort			:= TRUE;
		END_IF
		(*====================================*)
    20080:
       Robot.M_ResetRobotAbsMove(UseA,UseB);; // Clear command 

        IF NOT Robot._DI1.Done THEN
			bRobotTimeOutIN := FALSE; // Edited by Jidien Kachu in 2025/10/09
            uiExecutingStep := 80000; 
        END_IF
		(* Edited by Jidien Kachu in 2025/10/09 *)

		bRobotTimeOutIN := TRUE;

		IF tonRobotTimeOut.Q THEN
			bRobotTimeOutIN := FALSE;
			strStatus :='FB_RobotRegionMove_FeedInConveyor_V2 Step 20080: Reset Robot timeout';


			_Error:=TRUE;
		END_IF	
		(*===================================*)
	
	30000:
			IF Get THEN
				IF   Robot._DI1.ClampA_Open AND Robot._DI1.ClampB_Open THEN
					uiExecutingStep := 31000;
				ELSE
					_Error	  := TRUE;
					strStatus := 'FB_RobotRegionMove_FeedInConveyor_V2 Step 30000: Clamp not open';
				END_IF
			ELSE
				IF NOT Robot._DI1.ClampA_Open AND NOT Robot._DI1.ClampB_Open THEN
					uiExecutingStep := 31000;
				ELSE
					_Error	  := TRUE;
					strStatus := 'FB_RobotRegionMove_FeedInConveyor_V2 Step 30000: Clamp is open';
				END_IF 
			END_IF		
		
		
    31000: // Both Clamps
        		
		
		  CASE uiBothStep OF
           		0://	
					BoxReady_1st := FALSE;
					BoxReady_2nd := FALSE;
					CASE Address_A OF
						1,2:
							uiBothStep:=1000;
						
						3: 
							uiBothStep:=100;
					END_CASE				
				100:	
					tonDelay.IN := FALSE;
					LowerConveyor.M_MoveBackward();
					bTimeOutIN:=FALSE;
					IF (NOT Input.bLowCV_BoxArrived_Sensor) AND  Input.bLowCV_2ndBoxGap_Sensor THEN
						uiBothStep:=150;
					END_IF
					bTimeOutIN:=TRUE;
					IF tonTimeOut.Q=TRUE OR Robot._DI1.Error THEN
						strStatus 		:= 'FB_RobotRegionMove_FeedInConveyor_V2 Step 31000: Empty conveyor timeout';
						Error 			:= TRUE;
						uiResumeStep	:= 31000;
						uiLastBothStep  := 0; //Edited by Jidien Kachu in 2025/10/09
						uiAbortingStep  := 0;//Edited by Jidien Kachu in 2025/10/14
						_Abort:=TRUE;
					END_IF	
					
				150:
					tonDelay.IN := TRUE;
					IF tonDelay.Q THEN
						uiBothStep:=200;
					END_IF		
				200:
					tonDelay.IN := FALSE;
					LowerConveyor.M_MotorStop();
					uiBothStep:=300;
				
				300:
					IF 	LowerConveyor.InStopped THEN
						bTimeOutIN:=FALSE;
						BoxReady_1st:=TRUE;
						uiBothStep:=1000;
					END_IF
					bTimeOutIN:=TRUE;
					IF tonTimeOut.Q=TRUE OR Robot._DI1.Error THEN
						strStatus :='FB_RobotRegionMove_FeedInConveyor_V2 Step 31000: Stop conveyor timeout';

						(* Edited by Jidien Kachu in 2025/10/09 *)
//						_Error:=TRUE;
						uiResumeStep := 31000;
						uiLastBothStep := 200;
						uiAbortingStep := 0;//Edited by Jidien Kachu in 2025/10/14
						_Abort := TRUE;
						(*====================================*)
					END_IF		

				1000:
							CASE Address_A OF							
						1:
								IF bCheckUpperCV_ServiceDone AND Input.bUpCV_Block1Detect_Sensor THEN
										BoxReady_1st := TRUE;
								END_IF
						2:
								IF bCheckUpperCV_ServiceDone AND Input.bUpCV_BoxArrived_Sensor THEN
										BoxReady_1st := TRUE;
								END_IF
						END_CASE
						
						IF Robot._DI1.Notification THEN
							uiBothStep:=2000;
						END_IF
						
				2000:

						CASE Address_B OF
						1,2:
							uiBothStep:=9000;						
						3: 
							uiBothStep:=3000;
					END_CASE	
				
				3000:	
					tonDelay.IN := FALSE;
					LowerConveyor.M_MoveBackward();
					IF (NOT Input.bLowCV_BoxArrived_Sensor) AND Input.bLowCV_2ndBoxGap_Sensor THEN
						bTimeOutIN:=FALSE;
						uiBothStep:=3100;
					END_IF
					bTimeOutIN:=TRUE;
					IF tonTimeOut.Q=TRUE OR Robot._DI1.Error THEN
						strStatus := 'FB_RobotRegionMove_FeedInConveyor_V2 Step 31000: Empty conveyor timeout';
						uiResumeStep:=31000;
						uiLastBothStep := 2000; // Edited by Jidien Kachu in 2025/10/09
						uiAbortingStep := 0;//Edited by Jidien Kachu in 2025/10/14
						_Abort:=TRUE;
					END_IF	
					
				3100:
					
					tonDelay.IN := TRUE;
					IF tonDelay.Q THEN
						uiBothStep:=3200;
					END_IF		
				3200:
					tonDelay.IN := FALSE;
					LowerConveyor.M_MotorStop();
					uiBothStep:=3300;
				
				3300:
					IF 	LowerConveyor.InStopped THEN
						bTimeOutIN:=FALSE;
						BoxReady_2nd:=TRUE;
						uiBothStep:=9999;
					END_IF
					bTimeOutIN:=TRUE;
					IF tonTimeOut.Q=TRUE OR Robot._DI1.Error THEN
						strStatus :='FB_RobotRegionMove_FeedInConveyor_V2 Step 31000: Stop conveyor timeout';




						(* Edited by Jidien Kachu in 2025/10/09 *)
//						_Error:=TRUE;
						uiResumeStep := 31000;
						uiLastBothStep := 3200;
						uiAbortingStep := 0;//Edited by Jidien Kachu in 2025/10/14
						_Abort := TRUE;
						(*====================================*)
					END_IF		
				9000:
							CASE Address_B OF							
						1:
								IF bCheckUpperCV_ServiceDone AND Input.bUpCV_Block1Detect_Sensor THEN
									BoxReady_2nd := TRUE;
								END_IF
						
						2:
								IF bCheckUpperCV_ServiceDone AND Input.bUpCV_BoxArrived_Sensor THEN
									BoxReady_2nd := TRUE;
								END_IF

						END_CASE
				
				9999: //Wait		
        // wait reset
        END_CASE

       	  // Robot Abs move
           		 Robot.M_StartRobotAbsMove( GetBox:=Get,
											UseClampA:=UseA,
											UseClampB:=UseB,
											Area:=Area,
											ClampA_Address:=Address_A,
											ClampB_Address:=Address_B,
											BoxReady_1:=BoxReady_1st,
											BoxReady_2:=BoxReady_2nd);	
		
		
        IF Robot._DI1.Done THEN

			bRobotTimeOutIN := FALSE; //Edited by Jidien Kachu in 2025/10/09
            uiExecutingStep := 30080;
        END_IF
		(* Edited by Jidien Kachu in 2025/10/09*)

		bRobotTimeOutIN := TRUE;

		IF tonRobotTimeOut.Q THEN

			bRobotTimeOutIN := FALSE;
			uiResumeStep	:= 31000;
		(*===================================*)
			strStatus := 'FB_RobotRegionMove_FeedInConveyor_V2 Step 31000: Robot Abs move timeout'; 
			_Abort			:= TRUE;
		END_IF
		IF Robot.Error THEN
			bRobotTimeOutIN	:= FALSE;
			uiResumeStep	:= 31000;
			strStatus		:= CONCAT('FB_RobotRegionMove_FeedInConveyor_V2',robot.ErrMsg);
			_Abort			:= TRUE;
		END_IF
    30080: // Check robot command is clear
        
        Robot.M_ResetRobotAbsMove(UseA,UseB);

        IF NOT Robot._DI1.Done THEN
			(* Edited by Jidien Kachu in 2025/10/09*)

			bRobotTimeOutIN := FALSE;
            uiExecutingStep := 80000; // go to place step
        END_IF    

		bRobotTimeOutIN := TRUE;

		IF tonRobotTimeOut.Q THEN
			(*===================================*)
			strStatus :='FB_RobotRegionMove_FeedInConveyor_V2 Step 31080: Stop Robot timeout';


			_Error:=TRUE;
		END_IF	
   
		
	80000:
		IF UseA THEN
			CASE Address_A OF
			1:
//				IF Input.bUpCV_BoxArrived_Sensor.P_SignalState THEN
//					strStatus :='Box not taken on F1';
//					_Error:=TRUE;
//				END_IF
				 uiExecutingStep :=99000;
			2:	
//				IF Input.bUpCV_Block1Detect_Sensor.P_SignalState THEN
//					strStatus :='Box not taken on F2';
//					_Error:=TRUE;
//				END_IF	
					uiExecutingStep :=99000;

			3:
				uiExecutingStep :=81000;			
			END_CASE
		END_IF
		IF UseB THEN
			CASE Address_B OF
			1:
//				IF Input.bUpCV_BoxArrived_Sensor.P_SignalState THEN
//					strStatus :='Box not taken on F1';
//					_Error:=TRUE;
//				END_IF
				 uiExecutingStep :=99000;
			2:	
//				IF Input.bUpCV_Block1Detect_Sensor.P_SignalState THEN
//					strStatus :='Box not taken on F2';
//					_Error:=TRUE;
//				END_IF	
					uiExecutingStep :=99000;

			3:
				uiExecutingStep :=81000;			
			END_CASE
		END_IF
		
	81000:
			LowerConveyor.M_MoveBackward();
			bTimeOutIN:=FALSE;
			IF (NOT Input.bLowCV_BoxArrived_Sensor) AND ( Input.bLowCV_2ndBoxGap_Sensor) THEN
						uiExecutingStep:=81100;
			END_IF
			bTimeOutIN:=TRUE;
			IF tonTimeOut.Q=TRUE OR Robot._DI1.Error THEN
				strStatus :='FB_RobotRegionMove_FeedInConveyor_V2 Step 81000: Empty conveyor timeout';


				(* Edited by Jidien Kachu in 2025/10/09 *)

				uiResumeStep := 81000;
				uiAbortingStep := 0;//Edited by Jidien Kachu in 2025/10/14
				_Abort := TRUE;
				(*====================================*)
			END_IF	
	81100:		
			LowerConveyor.M_MotorStop();
			uiExecutingStep:=81200;
				
	81200:
			IF 	LowerConveyor.InStopped THEN
				bTimeOutIN:=FALSE;
				uiExecutingStep:=99000;
			END_IF
			bTimeOutIN:=TRUE;
			IF tonTimeOut.Q=TRUE OR Robot._DI1.Error THEN
				strStatus :='FB_RobotRegionMove_FeedInConveyor_V2 Step 81200: Stop conveyor timeout';


				(* Edited by Jidien Kachu in 2025/10/09 *)

				uiResumeStep := 81100;
				uiAbortingStep := 0;//Edited by Jidien Kachu in 2025/10/14
				_Abort := TRUE;
				(*====================================*)
			END_IF		
					
    99000: 	  // process done
          Status    := 'FB_RobotRegionMove_FeedInConveyor_V2 Step 99000: Process completed';
      	  _Executed := TRUE;
		  uiBothStep:= 0; //Edited by Jidien Kachu in 2025/10/14
		  uiSingleClampStep := 0;//Edited by Jidien Kachu in 2025/10/14
END_CASE

// ================= STATE Control ==================
IF NOT Execute THEN
    eState 	:= STATE_RESETTING;
ELSIF _Error THEN
    eState	:= STATE_ERROR;
ELSIF _Abort THEN
	eSTATE	:= STATE_ABORTING;
ELSIF _Executed THEN
    eState 					:= STATE_DONE;
	uiLastBothStep 			:= 0; //Edited by Jidien Kachu in 2025/10/14
	uiLastSingleClampStep 	:= 0; //Edited by Jidien Kachu in 2025/10/14
END_IF
END_METHOD

METHOD  M_STATE_RESETTING
VAR_INPUT
END_VAR
// Done := false 更改到Dormant 清除確保，上位檢查到done 後可以直接下Execute

CASE uiResettingStep OF

	0:
		tonDelay.IN := FALSE;
		bTimeOutIN:=FALSE;
		Robot.M_ResetAllCommand();
		Robot.M_ResetRobotAbsMove(TRUE,TRUE);
		uiResettingStep:=100;
		tonRobotTimeOut.IN := FALSE;

	100:

		LowerConveyor.M_MotorStop();
		uiResettingStep:=9999;
	9999:
//		Done := FALSE;
//		Busy := FALSE;
		_ResetCompleted:=TRUE;
END_CASE
IF _ResetCompleted THEN
	eSTATE:=STATE_DORMANT;
END_IF
END_METHOD

END_FUNCTION_BLOCK

// ---- Library/20_MachineUnits/21_StorageArea/Service_Robot/FB_RobotRegionMove_PullOutConveyor.TcPOU
FUNCTION_BLOCK FB_RobotRegionMove_PullOutConveyor EXTENDS FB_ObjectBase_V2 IMPLEMENTS IBasicElement
VAR_INPUT
    Robot     				: REFERENCE TO FB_FanucRobot_Basic_V2;
	PullOutConveyor 		: REFERENCE TO FB_PullOutConveyorAction; // Allocated area pull out conveyor
    Info	  				: ST_RobotRegionMove_Info;
	Stop	  : BOOL;
END_VAR
VAR_OUTPUT
  // Status : ST_WareHouseWithRobotMove_Status;
END_VAR
VAR
	//_Abort		: BOOL;
	strStatus	: STRING;
	uiResumeStep : UINT;
	
	Area	: E_RobotArea:=E_RobotArea.PullOutConveyor;
	UseA 	: BOOL;
	UseB	: BOOL;
	
	Get 	:BOOL;
	tonTimeOut	:TON;
	_UniqueErrorCode :STRING;
	PreviousStrStatus : STRING;
	PreviousErrorCode : STRING;
	
	_bRetry		: BOOL;
END_VAR

SUPER^.A10_StateControl();
A00_BasicUnits();

ACTION A00_BasicUnits:
tonTimeOut(PT:=T#60S);
ErrorID:=2230;
END_ACTION

METHOD M_CheckClampStatus : BOOL
VAR_INPUT
END_VAR
M_CheckClampStatus := FALSE;

IF NOT UseA AND NOT UseB THEN
	M_CheckClampStatus 	:= FALSE;
	strStatus 			:= 'FB_RobotRegionMove_PullOutConveyor: Wrong Command , Both Clammp not used';
	RETURN;
END_IF

IF UseA THEN
	IF Get THEN
		IF NOT Robot._DI1.ClampA_Open THEN
			M_CheckClampStatus  := FALSE;
			strStatus			:= 'FB_RobotRegionMove_PullOutConveyor: Robot Use A Clamp Get ,but Clamp not open ';
			RETURN;
		END_IF
	ELSE
		IF Robot._DI1.ClampA_Open THEN
			M_CheckClampStatus	:= FALSE;
			strStatus			:= 'FB_RobotRegionMove_PullOutConveyor: Robot Use A Clamp Place ,but Clamp open';
			RETURN;
		END_IF
	END_IF
END_IF
IF UseB THEN
	IF Get THEN
		IF NOT Robot._DI1.ClampB_Open THEN
			M_CheckClampStatus  := FALSE;
			strStatus			:= 'FB_RobotRegionMove_PullOutConveyor: Robot Use B Clamp Get ,but Clamp not open ';
			RETURN;
		END_IF
	ELSE
		IF Robot._DI1.ClampB_Open THEN
			M_CheckClampStatus	:= FALSE;
			strStatus			:= 'FB_RobotRegionMove_PullOutConveyor: Robot Use B Clamp Place ,but Clamp open';
			RETURN;
		END_IF
	END_IF
END_IF

M_CheckClampStatus := TRUE;
END_METHOD

METHOD M_CheckCommand : BOOL // True : Command is useful
VAR_INPUT
END_VAR
VAR
	
END_VAR
// Check command paremeter is correct
		
	THIS^.Get :=Info.Get;
	UseA :=Info.UseA;
	UseB :=Info.UseB;

	 // PullOut conveyor
		IF UseA AND (Info.A_Position<1 OR  Info.A_Position>2 )THEN
			strStatus:='FB_RobotRegionMove_PullOutConveyor: Wrong command ,Position A Not allow';
			M_CheckCommand:=FALSE;
			RETURN;				
		END_IF	
	
		IF UseB AND (Info.B_Position<1 OR  Info.B_Position>2 )THEN
			strStatus:='FB_RobotRegionMove_PullOutConveyor: Wrong command ,Position B Not allow';
			M_CheckCommand:=FALSE;
			RETURN;			
		END_IF
	



M_CheckCommand:=TRUE;
END_METHOD

METHOD M_CheckUnitsNotBusy : BOOL
VAR_INPUT
END_VAR
M_CheckUnitsNotBusy := true;
END_METHOD

METHOD M_CheckUnitsReady : BOOL
VAR_INPUT
END_VAR
M_CheckUnitsReady := true;
END_METHOD

METHOD  M_STATE_ABORTED
VAR_INPUT
END_VAR
IF NOT _bRetry THEN
	ERROR 	:= TRUE;
	Busy    := FALSE;
	Aborted := TRUE;
	Status  := strStatus;
	UniqueErrorCode := _UniqueErrorCode;
	_AbortCompleted := FALSE;
	uiAbortingStep	:= 0;
END_IF

IF reset THEN
	_bRetry := TRUE;
	Error	:= FALSE;
	Aborted	:= FALSE;
END_IF

IF NOT Execute THEN
	eSTATE:=STATE_RESETTING;
END_IF
IF Execute AND _bRetry AND NOT robot._DI1.Error AND NOT Robot.Halt THEN
	status	:= '';
	PreviousStrStatus := strStatus;
	PreviousErrorCode := _UniqueErrorCode;
	uiExecutingStep :=uiResumeStep;
	
	IF GVL_ADS.MachineState <>E_MachineState.Error THEN
		eSTATE:=STATE_EXECUTING;
	END_IF
END_IF
END_METHOD

METHOD  M_STATE_ABORTING
VAR_INPUT
END_VAR
CASE uiAbortingStep OF
	0 :
			
			DAS_CoreSys.MachineControl.fbStorageArea.M_ResetSlides_FeedOut();
			tonTimeOut.IN:= FALSE;
			_Abort 		 := FALSE;
			_bRetry		 := FALSE;
			IF strStatus = PreviousStrStatus THEN
				_UniqueErrorCode :=PreviousErrorCode;
			END_IF
			uiAbortingStep := 100;
	100:
			IF Robot._DI1.Error THEN
				uiAbortingStep := 200;
			ELSE
				uiAbortingStep := 9999;
			END_IF
	200:		
			 IF DAS_CoreSys.MachineControl.M_RobotResetCmd() THEN
				 uiAbortingStep := 300;
			 END_IF
	300:
			IF DAS_CoreSys.MachineControl.M_RobotStartCmd() THEN
				 uiAbortingStep := 400;
			 END_IF 
	400:
			IF Robot._DI1.Error THEN
		 		uiAbortingStep := 200;
			ELSE
				uiAbortingStep := 9999;
			END_IF
	9999:	
			_AbortCompleted:=TRUE;
END_CASE

IF _AbortCompleted THEN	
	eSTATE :=STATE_ABORTED;
END_IF
END_METHOD

METHOD  M_STATE_DONE
VAR_INPUT
END_VAR
Busy   := FALSE;
_Error := Error := FALSE;
_Abort := Abort := FALSE;
Done   := TRUE;

IF NOT Execute THEN
    eState := STATE_RESETTING;
END_IF
END_METHOD

METHOD  M_STATE_DORMANT
VAR_INPUT
END_VAR
// Clear FB output
Busy            := FALSE;
Done            := FALSE;
Aborted         := FALSE;
Error           := FALSE;
ErrorID         := 0;
Status          := '';
_ResetCompleted := FALSE;
_Error          := FALSE;
_Executed       := FALSE;

tonTimeOut.IN:=FALSE;
strStatus :='No Error';
uiExecutingStep :=uiResettingStep :=uiResumeStep :=0;
PreviousStrStatus			 :='';
PreviousErrorCode			 :='';
uiAbortingStep := 0;
_AbortCompleted:= FALSE;
_bRetry	:= FALSE;


// Wait Execute command
IF Execute AND NOT stop THEN
    eState := STATE_EXECUTING;
END_IF
END_METHOD

METHOD  M_STATE_ERROR
VAR_INPUT
END_VAR
ERROR   :=TRUE;
Busy	:=FALSE;
Status := strStatus;
UniqueErrorCode:=_UniqueErrorCode;
IF NOT Execute THEN	
eSTATE:=STATE_RESETTING;
END_IF
END_METHOD

METHOD  M_STATE_EXECUTING
VAR_INPUT
END_VAR
VAR_INST
	BoxReady_1st : BOOL;
	BoxReady_2nd : BOOL;
    uiBothStep : UINT;
    uiSingleClampStep : UINT;	
	Area : E_RobotArea;
	Address_A : INT;
	Address_B : INT;
END_VAR
VAR
	WareHouse: INT;
	LowerConveyor: INT;
END_VAR
// Set Busy active edit by johnson
Busy := TRUE;

IF THIS^.Stop THEN // Pending the timeout when Stop signal occur
    tonTimeout.IN := FALSE;
END_IF

// Service Process
CASE uiExecutingStep OF
    0:
        // Clear variable
        uiBothStep := 0;
        uiSingleClampStep := 0;
        BoxReady_1st := 0;
        BoxReady_2nd := 0;
        tonTimeOut.IN := FALSE;

        // Check command
        IF M_CheckCommand() THEN
            uiExecutingStep := 10;
        ELSE
            _Error := TRUE;
        END_IF
    10:
        // Start process, check units first
        IF M_CheckUnitsReady() THEN
            uiExecutingStep := 20;
        END_IF
    20:
        // CHeck units not busy state
        IF M_CheckUnitsNotBusy() THEN
            uiExecutingStep := 30;
        END_IF
	30:
		IF M_CheckClampStatus() THEN
			uiExecutingStep := 1000;
		ELSE
			_Abort := TRUE;
		END_IF

    1000:
        // Read   coordinate
        Area := THIS^.Area;
        Address_A := LREAL_TO_INT(Info.A_Position);
        Address_B := LREAL_TO_INT(Info.B_Position);
        DAS_CoreSys.MachineControl.fballocatearea.M_GetPulloutAccess(ControlAccess := E_RoundBeltControlAccess.FanucRobot);

        IF UseA AND NOT UseB THEN
            //Only clampA
            uiExecutingStep := 10000;
        ELSIF NOT UseA AND UseB THEN
            //Only ClampB 
            uiExecutingStep := 20000;
        ELSIF UseA AND UseB THEN
            //Both Clamps
            uiExecutingStep := 30000;
        END_IF

    10000: // Only ClampA 
        IF NOT Robot._DI1.Done THEN

            IF Get THEN // Get box job

                CASE Address_A OF
                    1:
                        DAS_CoreSys.MachineControl.fballocatearea
                            .M_StartStoragePulloutAction(CommandType := E_PullOutConveyorCommandType.SlideB_FeedIn_Ext,
                                                         CV_BackwardTIme := T#0S,
                                                         CV_ForwardTime := T#0S);
                    2:
                        DAS_CoreSys.MachineControl.fballocatearea
                            .M_StartStoragePulloutAction(CommandType := E_PullOutConveyorCommandType.SlideA_FeedIn_Ext,
                                                         CV_BackwardTIme := T#0S,
                                                         CV_ForwardTime := T#0S);
                END_CASE

            ELSE
                CASE Address_A OF
                    1:
                        DAS_CoreSys.MachineControl.fballocatearea
                            .M_StartStoragePulloutAction(CommandType := E_PullOutConveyorCommandType.SlideB_FeedOut_Ext,
                                                         CV_BackwardTIme := T#2S,
                                                         CV_ForwardTime := T#0S);

                    2:
                        DAS_CoreSys.MachineControl.fballocatearea
                            .M_StartStoragePulloutAction(CommandType := E_PullOutConveyorCommandType.SlideA_FeedOut_Ext,
                                                         CV_BackwardTIme := T#2S,
                                                         CV_ForwardTime := T#0S);
                END_CASE

            END_IF

            // Robot Abs move
            Robot.M_StartRobotAbsMove(GetBox := Get,
                                      UseClampA := UseA,
                                      UseClampB := UseB,
                                      Area := Area,
                                      ClampA_Address := Address_A,
                                      ClampB_Address := Address_B,
                                      BoxReady_1 := DAS_CoreSys.MachineControl.fballocatearea.fbPulloutCv.Done,
                                      BoxReady_2 := FALSE);

        ELSE
            tonTimeOut.IN := FALSE;
            uiExecutingStep := 10080;
        END_IF

        IF DAS_CoreSys.MachineControl.fballocatearea.fbPulloutCv.Error THEN
            DAS_CoreSys.MachineControl.fballocatearea.M_StopStoragePulloutAction();
            uiResumeStep := 10000;
            _Abort := TRUE;
            strStatus := 'FB_RobotRegionMove_PullOutConveyor Step 10000: Pullout CV error';


        END_IF

        tonTimeOut.IN := TRUE;

        IF tonTimeOut.Q = TRUE THEN
            tonTimeOut.IN := FALSE;
            strStatus 	  := 'FB_RobotRegionMove_PullOutConveyor Step 10000: Robot Move timeout';
            uiResumeStep := 10000;
            _Abort := TRUE;
        END_IF
    10080:
        Robot.M_ResetRobotAbsMove(UseA, UseB); // Clear command and go to place box
        DAS_CoreSys.MachineControl.fballocatearea.M_StopStoragePulloutAction();
        tonTimeOut.IN := TRUE;

        IF NOT Robot._DI1.Done THEN
            tonTimeOut.IN := FALSE;
            uiExecutingStep := 99000;
        END_IF

        IF tonTimeOut.Q = TRUE THEN
            strStatus := 'FB_RobotRegionMove_PullOutConveyor Step 10080: Reset Robot timeout';




            _Error := TRUE;
        END_IF

    20000: // Only ClampB
        IF NOT Robot._DI1.Done THEN

            IF Get THEN // Get box job

                CASE Address_B OF
                    1:
                        DAS_CoreSys.MachineControl.fballocatearea
                            .M_StartStoragePulloutAction(CommandType := E_PullOutConveyorCommandType.SlideB_FeedIn_Ext,
                                                         CV_BackwardTIme := T#2S,
                                                         CV_ForwardTime := T#0S);

                    2:
                        DAS_CoreSys.MachineControl.fballocatearea
                            .M_StartStoragePulloutAction(CommandType := E_PullOutConveyorCommandType.SlideA_FeedIn_Ext,
                                                         CV_BackwardTIme := T#2S,
                                                         CV_ForwardTime := T#0S);
                END_CASE

            ELSE
                CASE Address_B OF
                    1:
                        DAS_CoreSys.MachineControl.fballocatearea
                            .M_StartStoragePulloutAction(CommandType := E_PullOutConveyorCommandType.SlideB_FeedOut_Ext,
                                                         CV_BackwardTIme := T#2S,
                                                         CV_ForwardTime := T#0S);

                    2:
                        DAS_CoreSys.MachineControl.fballocatearea
                            .M_StartStoragePulloutAction(CommandType := E_PullOutConveyorCommandType.SlideA_FeedOut_Ext,
                                                         CV_BackwardTIme := T#2S,
                                                         CV_ForwardTime := T#0S);
                END_CASE

            END_IF

            // Robot Abs move
            Robot.M_StartRobotAbsMove(GetBox := Get,
                                      UseClampA := UseA,
                                      UseClampB := UseB,
                                      Area := Area,
                                      ClampA_Address := Address_A,
                                      ClampB_Address := Address_B,
                                      BoxReady_1 := FALSE,
                                      BoxReady_2 := DAS_CoreSys.MachineControl.fballocatearea.fbPulloutCV.Done);

        ELSE
            tonTimeOut.IN := FALSE;
            uiExecutingStep := 20080;
        END_IF

        IF DAS_CoreSys.MachineControl.fballocatearea.fbPulloutCv.Error THEN
            DAS_CoreSys.MachineControl.fballocatearea.M_StopStoragePulloutAction();
            uiResumeStep := 20000;
            _Abort := TRUE;
            strStatus := 'FB_RobotRegionMove_PullOutConveyor Step 20000: Feed box timeout';


        END_IF

        tonTimeOut.IN := TRUE;

        IF tonTimeOut.Q = TRUE THEN
            tonTimeOut.IN := FALSE;
            strStatus := 'FB_RobotRegionMove_PullOutConveyor Step 20000: Robot Move timeout';
            uiResumeStep := 20000;
            _Abort := TRUE;
        END_IF
    20080:
        Robot.M_ResetRobotAbsMove(UseA, UseB);
        DAS_CoreSys.MachineControl.fballocatearea.M_StopStoragePulloutAction();
        ; // Clear command 

        IF NOT Robot._DI1.Done THEN
            uiExecutingStep := 99000;
        END_IF

        tonTimeOut.IN := TRUE;

        IF tonTimeOut.Q = TRUE THEN
            strStatus := 'FB_RobotRegionMove_PullOutConveyor Step 20080: Reset Robot timeout';


            _Error := TRUE;
        END_IF
    30000: // Both Clamps

        CASE uiBothStep OF
            0: //	
                BoxReady_1st := FALSE;
                BoxReady_2nd := FALSE;

                uiBothStep := 1000;

            1000:
                IF Get THEN // Get box job

                    CASE Address_A OF
                        1:
                            DAS_CoreSys.MachineControl.fballocatearea
                                .M_StartStoragePulloutAction(CommandType := E_PullOutConveyorCommandType.SlideB_FeedIn_Ext,
                                                             CV_BackwardTIme := T#0S,
                                                             CV_ForwardTime := T#0S);
                        2:
                            DAS_CoreSys.MachineControl.fballocatearea
                                .M_StartStoragePulloutAction(CommandType := E_PullOutConveyorCommandType.SlideA_FeedIn_Ext,
                                                             CV_BackwardTIme := T#0S,
                                                             CV_ForwardTime := T#0S);
                    END_CASE

                ELSE
                    CASE Address_A OF
                        1:
                            DAS_CoreSys.MachineControl.fballocatearea
                                .M_StartStoragePulloutAction(CommandType := E_PullOutConveyorCommandType.SlideB_FeedOut_Ext,
                                                             CV_BackwardTIme := T#2S,
                                                             CV_ForwardTime := T#0S);

                        2:
                            DAS_CoreSys.MachineControl.fballocatearea
                                .M_StartStoragePulloutAction(CommandType := E_PullOutConveyorCommandType.SlideA_FeedOut_Ext,
                                                             CV_BackwardTIme := T#2S,
                                                             CV_ForwardTime := T#0S);
                    END_CASE

                END_IF

                uiBothStep := 1100;
            1100:
                IF DAS_CoreSys.MachineControl.fballocatearea.fbPulloutCv.Done THEN
                    DAS_CoreSys.MachineControl.fballocatearea.M_StopStoragePulloutAction();
                    BoxReady_1st := TRUE;
                    uiBothStep := 2000;
                END_IF

                IF DAS_CoreSys.MachineControl.fballocatearea.fbPulloutCv.Error THEN
                    DAS_CoreSys.MachineControl.fballocatearea.M_StopStoragePulloutAction();
                    uiResumeStep := 30000;
                    uiBothStep := 1000;
                    _Abort := TRUE;
                    strStatus := 'FB_RobotRegionMove_PullOutConveyor Step 30000: Feed box timeout';


                END_IF

            2000:
                IF Robot._DI1.Notification THEN
                    uiBothStep := 3000;
                END_IF
            3000:

                IF Get THEN // Get box job

                    CASE Address_B OF
                        1:
                            DAS_CoreSys.MachineControl.fballocatearea
                                .M_StartStoragePulloutAction(CommandType := E_PullOutConveyorCommandType.SlideB_FeedIn_Ext,
                                                             CV_BackwardTIme := T#0S,
                                                             CV_ForwardTime := T#0S);
                        2:
                            DAS_CoreSys.MachineControl.fballocatearea
                                .M_StartStoragePulloutAction(CommandType := E_PullOutConveyorCommandType.SlideA_FeedIn_Ext,
                                                             CV_BackwardTIme := T#0S,
                                                             CV_ForwardTime := T#0S);
                    END_CASE

                ELSE
                    CASE Address_B OF
                        1:
                            DAS_CoreSys.MachineControl.fballocatearea
                                .M_StartStoragePulloutAction(CommandType := E_PullOutConveyorCommandType.SlideB_FeedOut_Ext,
                                                             CV_BackwardTIme := T#2S,
                                                             CV_ForwardTime := T#0S);

                        2:
                            DAS_CoreSys.MachineControl.fballocatearea
                                .M_StartStoragePulloutAction(CommandType := E_PullOutConveyorCommandType.SlideA_FeedOut_Ext,
                                                             CV_BackwardTIme := T#2S,
                                                             CV_ForwardTime := T#0S);
                    END_CASE
                END_IF

